LIN {X 0,Y 347.087,Z 840.961,A -85,B 0,C 180,E1 20651.677,E2 20651.677} C_VEL
LIN {X 0,Y 346.368,Z 839.475,A -85,B 0,C 180,E1 20653.232,E2 20653.232} C_VEL
LIN {X 0,Y 343.386,Z 836.917,A -85,B 0,C 180,E1 20663.758,E2 20663.758} C_VEL
LIN {X 0,Y 344.875,Z 838.107,A -85,B 0,C 180,E1 20672.864,E2 20672.864} C_VEL
LIN {X 0,Y 348.52,Z 840.648,A -85,B 0,C 180,E1 20679.253,E2 20679.253} C_VEL
LIN {X 0,Y 352.329,Z 846.298,A -85,B 0,C 180,E1 20684.292,E2 20684.292} C_VEL
LIN {X 0,Y 354.573,Z 848.436,A -85,B 0,C 180,E1 20686.475,E2 20686.475} C_VEL
LIN {X 0,Y 359.696,Z 854.398,A -85,B 0,C 180,E1 20690.882,E2 20690.882} C_VEL
LIN {X 0,Y 364.724,Z 861.307,A -85,B 0,C 180,E1 20694.66,E2 20694.66} C_VEL
LIN {X 0,Y 374.327,Z 875.302,A -85,B 0,C 180,E1 20700.736,E2 20700.736} C_VEL
LIN {X 0,Y 387.121,Z 895.572,A -85,B 0,C 180,E1 20707.425,E2 20707.425} C_VEL
LIN {X 0,Y 401.281,Z 919.676,A -85,B 0,C 180,E1 20713.739,E2 20713.739} C_VEL
LIN {X 0,Y 415.418,Z 946.976,A -85,B 0,C 180,E1 20719.523,E2 20719.523} C_VEL
LIN {X 0,Y 429.203,Z 977.889,A -85,B 0,C 180,E1 20724.99,E2 20724.99} C_VEL
LIN {X 0,Y 433.479,Z 989.391,A -85,B 0,C 180,E1 20726.807,E2 20726.807} C_VEL
LIN {X 0,Y 418.447,Z 1036.021,A -85,B 0,C 180,E1 20729.455,E2 20729.455} C_VEL
LIN {X 0,Y 400.123,Z 1083.411,A -85,B 0,C 180,E1 20733.256,E2 20733.256} C_VEL
LIN {X 0,Y 383.119,Z 1122.716,A -85,B 0,C 180,E1 20737.596,E2 20737.596} C_VEL
LIN {X 0,Y 366.033,Z 1159.658,A -85,B 0,C 180,E1 20743.097,E2 20743.097} C_VEL
LIN {X 0,Y 351.513,Z 1190.56,A -85,B 0,C 180,E1 20749.344,E2 20749.344} C_VEL
LIN {X 0,Y 339.716,Z 1217.292,A -85,B 0,C 180,E1 20756.591,E2 20756.591} C_VEL
LIN {X 0,Y 331.936,Z 1238.037,A -85,B 0,C 180,E1 20764.364,E2 20764.364} C_VEL
LIN {X 0,Y 328.007,Z 1253.422,A -85,B 0,C 180,E1 20772.565,E2 20772.565} C_VEL
LIN {X 0,Y 326.864,Z 1261.496,A -85,B 0,C 180,E1 20779.333,E2 20779.333} C_VEL
LIN {X 0,Y 326.773,Z 1264.976,A -85,B 0,C 180,E1 20784.683,E2 20784.683} C_VEL
LIN {X 0,Y 327.283,Z 1265.936,A -85,B 0,C 180,E1 20789.989,E2 20789.989} C_VEL
LIN {X 0,Y 327.033,Z 1263.961,A -85,B 0,C 180,E1 20795.291,E2 20795.291} C_VEL
LIN {X 0,Y 327.282,Z 1257.785,A -85,B 0,C 180,E1 20801.98,E2 20801.98} C_VEL
LIN {X 0,Y 328.698,Z 1247.276,A -85,B 0,C 180,E1 20808.76,E2 20808.76} C_VEL
LIN {X 0,Y 333.133,Z 1228.55,A -85,B 0,C 180,E1 20816.962,E2 20816.962} C_VEL
LIN {X 0,Y 340.815,Z 1205.172,A -85,B 0,C 180,E1 20824.41,E2 20824.41} C_VEL
LIN {X 0,Y 352.574,Z 1174.665,A -85,B 0,C 180,E1 20831.655,E2 20831.655} C_VEL
LIN {X 0,Y 369.605,Z 1134.827,A -85,B 0,C 180,E1 20838.789,E2 20838.789} C_VEL
LIN {X 0,Y 399.925,Z 1072.683,A -85,B 0,C 180,E1 20846.92,E2 20846.92} C_VEL
LIN {X 0,Y 420.751,Z 1039.494,A -85,B 0,C 180,E1 20850.42,E2 20850.42} C_VEL
LIN {X 0,Y 414.218,Z 1046.912,A -85,B 0,C 180,E1 20851.536,E2 20851.536} C_VEL
LIN {X 0,Y 403.987,Z 1058.605,A -85,B 0,C 180,E1 20852.711,E2 20852.711} C_VEL
LIN {X 0,Y 393.91,Z 1069.679,A -85,B 0,C 180,E1 20853.981,E2 20853.981} C_VEL
LIN {X 0,Y 366.198,Z 1101.609,A -85,B 0,C 180,E1 20861.35,E2 20861.35} C_VEL
LIN {X 0,Y 346.971,Z 1124.322,A -85,B 0,C 180,E1 20868.879,E2 20868.879} C_VEL
LIN {X 0,Y 332.663,Z 1141.932,A -85,B 0,C 180,E1 20877.586,E2 20877.586} C_VEL
LIN {X 0,Y 324.133,Z 1153.386,A -85,B 0,C 180,E1 20886.691,E2 20886.691} C_VEL
LIN {X 0,Y 320.638,Z 1158.38,A -85,B 0,C 180,E1 20893.627,E2 20893.627} C_VEL
LIN {X 0,Y 318.865,Z 1160.285,A -85,B 0,C 180,E1 20899.371,E2 20899.371} C_VEL
LIN {X 0,Y 318.24,Z 1159.445,A -85,B 0,C 180,E1 20908.345,E2 20908.345} C_VEL
LIN {X 0,Y 320.177,Z 1153.951,A -85,B 0,C 180,E1 20916.668,E2 20916.668} C_VEL
LIN {X 0,Y 323.485,Z 1144.81,A -85,B 0,C 180,E1 20924.477,E2 20924.477} C_VEL
LIN {X 0,Y 330.102,Z 1130.596,A -85,B 0,C 180,E1 20932.434,E2 20932.434} C_VEL
LIN {X 0,Y 341.206,Z 1109.637,A -85,B 0,C 180,E1 20940.43,E2 20940.43} C_VEL
LIN {X 0,Y 354.83,Z 1084.984,A -85,B 0,C 180,E1 20947.16,E2 20947.16} C_VEL
LIN {X 0,Y 371.931,Z 1052.972,A -85,B 0,C 180,E1 20953.488,E2 20953.488} C_VEL
LIN {X 0,Y 389.199,Z 1018.22,A -85,B 0,C 180,E1 20958.439,E2 20958.439} C_VEL
LIN {X 0,Y 402.022,Z 989.391,A -85,B 0,C 180,E1 20961.634,E2 20961.634} C_VEL
LIN {X 0,Y 397.777,Z 963.333,A -85,B 0,C 180,E1 20967.015,E2 20967.015} C_VEL
LIN {X 0,Y 391.25,Z 938.761,A -85,B 0,C 180,E1 20972.5,E2 20972.5} C_VEL
LIN {X 0,Y 383.479,Z 917.337,A -85,B 0,C 180,E1 20978.002,E2 20978.002} C_VEL
LIN {X 0,Y 374.105,Z 897.059,A -85,B 0,C 180,E1 20984.227,E2 20984.227} C_VEL
LIN {X 0,Y 364.994,Z 880.396,A -85,B 0,C 180,E1 20990.659,E2 20990.659} C_VEL
LIN {X 0,Y 356.896,Z 867.057,A -85,B 0,C 180,E1 20997.245,E2 20997.245} C_VEL
LIN {X 0,Y 351.496,Z 859.187,A -85,B 0,C 180,E1 21002.484,E2 21002.484} C_VEL
LIN {X 0,Y 348.543,Z 853.905,A -85,B 0,C 180,E1 21006.187,E2 21006.187} C_VEL
LIN {X 0,Y 344.933,Z 848.047,A -85,B 0,C 180,E1 21012.142,E2 21012.142} C_VEL
LIN {X 0,Y 341.412,Z 844.833,A -85,B 0,C 180,E1 21022.14,E2 21022.14} C_VEL
LIN {X 0,Y 342.46,Z 845.304,A -85,B 0,C 180,E1 21030.967,E2 21030.967} C_VEL
LIN {X 0,Y 346.658,Z 848.318,A -85,B 0,C 180,E1 21039.063,E2 21039.063} C_VEL
LIN {X 0,Y 350.624,Z 854.035,A -85,B 0,C 180,E1 21044.381,E2 21044.381} C_VEL
LIN {X 0,Y 352.591,Z 856.228,A -85,B 0,C 180,E1 21046.368,E2 21046.368} C_VEL
LIN {X 0,Y 358.34,Z 863.911,A -85,B 0,C 180,E1 21051.519,E2 21051.519} C_VEL
LIN {X 0,Y 364.09,Z 871.747,A -85,B 0,C 180,E1 21055.711,E2 21055.711} C_VEL
LIN {X 0,Y 371.715,Z 882.573,A -85,B 0,C 180,E1 21060.438,E2 21060.438} C_VEL
LIN {X 0,Y 384.55,Z 903.458,A -85,B 0,C 180,E1 21067.385,E2 21067.385} C_VEL
LIN {X 0,Y 398.907,Z 928.625,A -85,B 0,C 180,E1 21073.974,E2 21073.974} C_VEL
LIN {X 0,Y 413.219,Z 957.636,A -85,B 0,C 180,E1 21080.049,E2 21080.049} C_VEL
LIN {X 0,Y 426.149,Z 988.884,A -85,B 0,C 180,E1 21085.549,E2 21085.549} C_VEL
LIN {X 0,Y 427.428,Z 992.49,A -85,B 0,C 180,E1 21086.118,E2 21086.118} C_VEL
LIN {X 0,Y 411.898,Z 1039.158,A -85,B 0,C 180,E1 21088.873,E2 21088.873} C_VEL
LIN {X 0,Y 393.65,Z 1085.05,A -85,B 0,C 180,E1 21092.623,E2 21092.623} C_VEL
LIN {X 0,Y 375.324,Z 1125.898,A -85,B 0,C 180,E1 21097.294,E2 21097.294} C_VEL
LIN {X 0,Y 358.404,Z 1161.367,A -85,B 0,C 180,E1 21102.774,E2 21102.774} C_VEL
LIN {X 0,Y 342.557,Z 1194.163,A -85,B 0,C 180,E1 21109.732,E2 21109.732} C_VEL
LIN {X 0,Y 330.876,Z 1219.831,A -85,B 0,C 180,E1 21117.202,E2 21117.202} C_VEL
LIN {X 0,Y 323.159,Z 1240.493,A -85,B 0,C 180,E1 21125.553,E2 21125.553} C_VEL
LIN {X 0,Y 319.856,Z 1253.989,A -85,B 0,C 180,E1 21133.522,E2 21133.522} C_VEL
LIN {X 0,Y 318.936,Z 1261.313,A -85,B 0,C 180,E1 21140.444,E2 21140.444} C_VEL
LIN {X 0,Y 319.149,Z 1264.519,A -85,B 0,C 180,E1 21147.275,E2 21147.275} C_VEL
LIN {X 0,Y 319.396,Z 1263.956,A -85,B 0,C 180,E1 21152.701,E2 21152.701} C_VEL
LIN {X 0,Y 319.221,Z 1259.367,A -85,B 0,C 180,E1 21159.525,E2 21159.525} C_VEL
LIN {X 0,Y 320.143,Z 1250.527,A -85,B 0,C 180,E1 21166.439,E2 21166.439} C_VEL
LIN {X 0,Y 323.154,Z 1235.77,A -85,B 0,C 180,E1 21174.064,E2 21174.064} C_VEL
LIN {X 0,Y 329.761,Z 1214.688,A -85,B 0,C 180,E1 21181.895,E2 21181.895} C_VEL
LIN {X 0,Y 340.513,Z 1186.665,A -85,B 0,C 180,E1 21189.562,E2 21189.562} C_VEL
LIN {X 0,Y 356.571,Z 1149.838,A -85,B 0,C 180,E1 21197.099,E2 21197.099} C_VEL
LIN {X 0,Y 379.459,Z 1102.791,A -85,B 0,C 180,E1 21204.273,E2 21204.273} C_VEL
LIN {X 0,Y 407.74,Z 1056.018,A -85,B 0,C 180,E1 21209.875,E2 21209.875} C_VEL
LIN {X 0,Y 411.948,Z 1050.22,A -85,B 0,C 180,E1 21210.575,E2 21210.575} C_VEL
LIN {X 0,Y 393.91,Z 1069.679,A -85,B 0,C 180,E1 21213.981,E2 21213.981} C_VEL
LIN {X 0,Y 383.621,Z 1080.519,A -85,B 0,C 180,E1 21215.383,E2 21215.383} C_VEL
LIN {X 0,Y 373.62,Z 1090.572,A -85,B 0,C 180,E1 21216.898,E2 21216.898} C_VEL
LIN {X 0,Y 348.296,Z 1118.195,A -85,B 0,C 180,E1 21224.912,E2 21224.912} C_VEL
LIN {X 0,Y 330.88,Z 1137.842,A -85,B 0,C 180,E1 21233.444,E2 21233.444} C_VEL
LIN {X 0,Y 319.47,Z 1151.446,A -85,B 0,C 180,E1 21242.71,E2 21242.71} C_VEL
LIN {X 0,Y 313.933,Z 1158.619,A -85,B 0,C 180,E1 21251.099,E2 21251.099} C_VEL
LIN {X 0,Y 311.719,Z 1161.251,A -85,B 0,C 180,E1 21256.907,E2 21256.907} C_VEL
LIN {X 0,Y 310.439,Z 1161.855,A -85,B 0,C 180,E1 21262.915,E2 21262.915} C_VEL
LIN {X 0,Y 310.489,Z 1160.35,A -85,B 0,C 180,E1 21269.119,E2 21269.119} C_VEL
LIN {X 0,Y 312.034,Z 1156.411,A -85,B 0,C 180,E1 21275.526,E2 21275.526} C_VEL
LIN {X 0,Y 314.99,Z 1148.284,A -85,B 0,C 180,E1 21283.171,E2 21283.171} C_VEL
LIN {X 0,Y 321.499,Z 1134.063,A -85,B 0,C 180,E1 21291.803,E2 21291.803} C_VEL
LIN {X 0,Y 331.447,Z 1115.81,A -85,B 0,C 180,E1 21299.382,E2 21299.382} C_VEL
LIN {X 0,Y 345.916,Z 1090.359,A -85,B 0,C 180,E1 21306.861,E2 21306.861} C_VEL
LIN {X 0,Y 361.451,Z 1062.441,A -85,B 0,C 180,E1 21312.786,E2 21312.786} C_VEL
LIN {X 0,Y 379.966,Z 1026.941,A -85,B 0,C 180,E1 21318.283,E2 21318.283} C_VEL
LIN {X 0,Y 395.881,Z 992.175,A -85,B 0,C 180,E1 21322.332,E2 21322.332} C_VEL
LIN {X 0,Y 391.593,Z 965.019,A -85,B 0,C 180,E1 21328.089,E2 21328.089} C_VEL
LIN {X 0,Y 385.246,Z 941.027,A -85,B 0,C 180,E1 21333.664,E2 21333.664} C_VEL
LIN {X 0,Y 377.827,Z 920.469,A -85,B 0,C 180,E1 21339.215,E2 21339.215} C_VEL
LIN {X 0,Y 368.976,Z 901.092,A -85,B 0,C 180,E1 21345.448,E2 21345.448} C_VEL
LIN {X 0,Y 360.705,Z 885.967,A -85,B 0,C 180,E1 21351.602,E2 21351.602} C_VEL
LIN {X 0,Y 353.28,Z 873.457,A -85,B 0,C 180,E1 21358.077,E2 21358.077} C_VEL
LIN {X 0,Y 348.747,Z 866.385,A -85,B 0,C 180,E1 21362.781,E2 21362.781} C_VEL
LIN {X 0,Y 345.909,Z 861.286,A -85,B 0,C 180,E1 21366.567,E2 21366.567} C_VEL
LIN {X 0,Y 342.565,Z 855.118,A -85,B 0,C 180,E1 21372.576,E2 21372.576} C_VEL
LIN {X 0,Y 339.4,Z 852.307,A -85,B 0,C 180,E1 21383.279,E2 21383.279} C_VEL
LIN {X 0,Y 340.932,Z 853.277,A -85,B 0,C 180,E1 21392.449,E2 21392.449} C_VEL
LIN {X 0,Y 344.532,Z 855.901,A -85,B 0,C 180,E1 21398.888,E2 21398.888} C_VEL
LIN {X 0,Y 348.882,Z 861.791,A -85,B 0,C 180,E1 21404.62,E2 21404.62} C_VEL
LIN {X 0,Y 355.837,Z 871.057,A -85,B 0,C 180,E1 21411.147,E2 21411.147} C_VEL
LIN {X 0,Y 361.762,Z 879.343,A -85,B 0,C 180,E1 21415.558,E2 21415.558} C_VEL
LIN {X 0,Y 368.908,Z 889.842,A -85,B 0,C 180,E1 21420.192,E2 21420.192} C_VEL
LIN {X 0,Y 380.831,Z 909.583,A -85,B 0,C 180,E1 21426.837,E2 21426.837} C_VEL
LIN {X 0,Y 394.818,Z 934.761,A -85,B 0,C 180,E1 21433.558,E2 21433.558} C_VEL
LIN {X 0,Y 408.62,Z 963.621,A -85,B 0,C 180,E1 21439.721,E2 21439.721} C_VEL
LIN {X 0,Y 420.981,Z 994.25,A -85,B 0,C 180,E1 21445.194,E2 21445.194} C_VEL
LIN {X 0,Y 421.256,Z 997.281,A -85,B 0,C 180,E1 21445.548,E2 21445.548} C_VEL
LIN {X 0,Y 404.179,Z 1045.484,A -85,B 0,C 180,E1 21448.513,E2 21448.513} C_VEL
LIN {X 0,Y 386.677,Z 1087.571,A -85,B 0,C 180,E1 21452.085,E2 21452.085} C_VEL
LIN {X 0,Y 367.331,Z 1129.407,A -85,B 0,C 180,E1 21457.017,E2 21457.017} C_VEL
LIN {X 0,Y 349.86,Z 1164.557,A -85,B 0,C 180,E1 21462.743,E2 21462.743} C_VEL
LIN {X 0,Y 334.671,Z 1195.273,A -85,B 0,C 180,E1 21469.517,E2 21469.517} C_VEL
LIN {X 0,Y 322.452,Z 1221.324,A -85,B 0,C 180,E1 21477.51,E2 21477.51} C_VEL
LIN {X 0,Y 315.188,Z 1240.426,A -85,B 0,C 180,E1 21485.625,E2 21485.625} C_VEL
LIN {X 0,Y 312.107,Z 1252.616,A -85,B 0,C 180,E1 21493.101,E2 21493.101} C_VEL
LIN {X 0,Y 311.126,Z 1259.993,A -85,B 0,C 180,E1 21500.202,E2 21500.202} C_VEL
LIN {X 0,Y 311.355,Z 1263.22,A -85,B 0,C 180,E1 21507.207,E2 21507.207} C_VEL
LIN {X 0,Y 311.589,Z 1262.619,A -85,B 0,C 180,E1 21512.768,E2 21512.768} C_VEL
LIN {X 0,Y 311.402,Z 1258.01,A -85,B 0,C 180,E1 21519.767,E2 21519.767} C_VEL
LIN {X 0,Y 312.394,Z 1249.057,A -85,B 0,C 180,E1 21526.859,E2 21526.859} C_VEL
LIN {X 0,Y 315.765,Z 1233.745,A -85,B 0,C 180,E1 21534.897,E2 21534.897} C_VEL
LIN {X 0,Y 323.109,Z 1211.687,A -85,B 0,C 180,E1 21543.164,E2 21543.164} C_VEL
LIN {X 0,Y 335.24,Z 1182.08,A -85,B 0,C 180,E1 21551.225,E2 21551.225} C_VEL
LIN {X 0,Y 353.239,Z 1143.875,A -85,B 0,C 180,E1 21558.984,E2 21558.984} C_VEL
LIN {X 0,Y 386.251,Z 1084.14,A -85,B 0,C 180,E1 21567.804,E2 21567.804} C_VEL
LIN {X 0,Y 401.734,Z 1062.211,A -85,B 0,C 180,E1 21570.426,E2 21570.426} C_VEL
LIN {X 0,Y 402.585,Z 1060.814,A -85,B 0,C 180,E1 21570.795,E2 21570.795} C_VEL
LIN {X 0,Y 373.62,Z 1090.572,A -85,B 0,C 180,E1 21576.898,E2 21576.898} C_VEL
LIN {X 0,Y 363.497,Z 1100.296,A -85,B 0,C 180,E1 21578.545,E2 21578.545} C_VEL
LIN {X 0,Y 353.613,Z 1109.353,A -85,B 0,C 180,E1 21580.331,E2 21580.331} C_VEL
LIN {X 0,Y 330.859,Z 1132.881,A -85,B 0,C 180,E1 21589.139,E2 21589.139} C_VEL
LIN {X 0,Y 315.905,Z 1148.961,A -85,B 0,C 180,E1 21598.629,E2 21598.629} C_VEL
LIN {X 0,Y 308.444,Z 1157.652,A -85,B 0,C 180,E1 21607.034,E2 21607.034} C_VEL
LIN {X 0,Y 304.794,Z 1161.898,A -85,B 0,C 180,E1 21614.35,E2 21614.35} C_VEL
LIN {X 0,Y 303.041,Z 1163.313,A -85,B 0,C 180,E1 21620.427,E2 21620.427} C_VEL
LIN {X 0,Y 302.488,Z 1162.504,A -85,B 0,C 180,E1 21626.715,E2 21626.715} C_VEL
LIN {X 0,Y 304.202,Z 1157.914,A -85,B 0,C 180,E1 21635.368,E2 21635.368} C_VEL
LIN {X 0,Y 307.365,Z 1149.485,A -85,B 0,C 180,E1 21643.489,E2 21643.489} C_VEL
LIN {X 0,Y 314.347,Z 1134.909,A -85,B 0,C 180,E1 21652.461,E2 21652.461} C_VEL
LIN {X 0,Y 324.691,Z 1116.522,A -85,B 0,C 180,E1 21660.166,E2 21660.166} C_VEL
LIN {X 0,Y 340.239,Z 1090.054,A -85,B 0,C 180,E1 21667.952,E2 21667.952} C_VEL
LIN {X 0,Y 357.448,Z 1059.64,A -85,B 0,C 180,E1 21674.285,E2 21674.285} C_VEL
LIN {X 0,Y 375.839,Z 1025.164,A -85,B 0,C 180,E1 21679.498,E2 21679.498} C_VEL
LIN {X 0,Y 389.627,Z 996.191,A -85,B 0,C 180,E1 21682.818,E2 21682.818} C_VEL
LIN {X 0,Y 386.32,Z 971.848,A -85,B 0,C 180,E1 21688.048,E2 21688.048} C_VEL
LIN {X 0,Y 380.76,Z 948.316,A -85,B 0,C 180,E1 21693.611,E2 21693.611} C_VEL
LIN {X 0,Y 374,Z 928.346,A -85,B 0,C 180,E1 21699.017,E2 21699.017} C_VEL
LIN {X 0,Y 365.792,Z 909.081,A -85,B 0,C 180,E1 21705.256,E2 21705.256} C_VEL
LIN {X 0,Y 357.652,Z 893.36,A -85,B 0,C 180,E1 21711.654,E2 21711.654} C_VEL
LIN {X 0,Y 350.277,Z 880.59,A -85,B 0,C 180,E1 21718.34,E2 21718.34} C_VEL
LIN {X 0,Y 346.244,Z 873.969,A -85,B 0,C 180,E1 21722.707,E2 21722.707} C_VEL
LIN {X 0,Y 344.049,Z 869.094,A -85,B 0,C 180,E1 21725.952,E2 21725.952} C_VEL
LIN {X 0,Y 340.256,Z 863.172,A -85,B 0,C 180,E1 21732.426,E2 21732.426} C_VEL
LIN {X 0,Y 337.277,Z 860.03,A -85,B 0,C 180,E1 21742.323,E2 21742.323} C_VEL
LIN {X 0,Y 338.315,Z 860.479,A -85,B 0,C 180,E1 21750.576,E2 21750.576} C_VEL
LIN {X 0,Y 342.401,Z 863.472,A -85,B 0,C 180,E1 21758.697,E2 21758.697} C_VEL
LIN {X 0,Y 346.957,Z 869.474,A -85,B 0,C 180,E1 21764.693,E2 21764.693} C_VEL
LIN {X 0,Y 353.516,Z 878.724,A -85,B 0,C 180,E1 21771.037,E2 21771.037} C_VEL
LIN {X 0,Y 359.005,Z 886.571,A -85,B 0,C 180,E1 21775.303,E2 21775.303} C_VEL
LIN {X 0,Y 366.202,Z 897.441,A -85,B 0,C 180,E1 21780.045,E2 21780.045} C_VEL
LIN {X 0,Y 377.529,Z 916.653,A -85,B 0,C 180,E1 21786.605,E2 21786.605} C_VEL
LIN {X 0,Y 390.304,Z 940.278,A -85,B 0,C 180,E1 21793.006,E2 21793.006} C_VEL
LIN {X 0,Y 403.47,Z 968.31,A -85,B 0,C 180,E1 21799.129,E2 21799.129} C_VEL
LIN {X 0,Y 415.487,Z 998.842,A -85,B 0,C 180,E1 21804.722,E2 21804.722} C_VEL
LIN {X 0,Y 397.445,Z 1049.215,A -85,B 0,C 180,E1 21807.946,E2 21807.946} C_VEL
LIN {X 0,Y 378.508,Z 1092.765,A -85,B 0,C 180,E1 21811.823,E2 21811.823} C_VEL
LIN {X 0,Y 360.009,Z 1131.337,A -85,B 0,C 180,E1 21816.538,E2 21816.538} C_VEL
LIN {X 0,Y 341.309,Z 1167.786,A -85,B 0,C 180,E1 21822.719,E2 21822.719} C_VEL
LIN {X 0,Y 326.235,Z 1197.103,A -85,B 0,C 180,E1 21829.561,E2 21829.561} C_VEL
LIN {X 0,Y 314.599,Z 1221.479,A -85,B 0,C 180,E1 21837.347,E2 21837.347} C_VEL
LIN {X 0,Y 307.118,Z 1240.519,A -85,B 0,C 180,E1 21845.878,E2 21845.878} C_VEL
LIN {X 0,Y 304.013,Z 1252.978,A -85,B 0,C 180,E1 21854.123,E2 21854.123} C_VEL
LIN {X 0,Y 303.306,Z 1259.571,A -85,B 0,C 180,E1 21861.393,E2 21861.393} C_VEL
LIN {X 0,Y 303.552,Z 1261.917,A -85,B 0,C 180,E1 21867.135,E2 21867.135} C_VEL
LIN {X 0,Y 303.789,Z 1261.304,A -85,B 0,C 180,E1 21872.839,E2 21872.839} C_VEL
LIN {X 0,Y 303.59,Z 1256.617,A -85,B 0,C 180,E1 21880.021,E2 21880.021} C_VEL
LIN {X 0,Y 304.642,Z 1247.636,A -85,B 0,C 180,E1 21887.302,E2 21887.302} C_VEL
LIN {X 0,Y 308.316,Z 1232.045,A -85,B 0,C 180,E1 21895.633,E2 21895.633} C_VEL
LIN {X 0,Y 316.164,Z 1209.949,A -85,B 0,C 180,E1 21904.065,E2 21904.065} C_VEL
LIN {X 0,Y 328.522,Z 1181.375,A -85,B 0,C 180,E1 21912.04,E2 21912.04} C_VEL
LIN {X 0,Y 348.658,Z 1141.259,A -85,B 0,C 180,E1 21920.351,E2 21920.351} C_VEL
LIN {X 0,Y 384.664,Z 1082.472,A -85,B 0,C 180,E1 21929.231,E2 21929.231} C_VEL
LIN {X 0,Y 394.161,Z 1069.933,A -85,B 0,C 180,E1 21930.852,E2 21930.852} C_VEL
LIN {X 0,Y 359.944,Z 1102.999,A -85,B 0,C 180,E1 21938.449,E2 21938.449} C_VEL
LIN {X 0,Y 353.613,Z 1109.353,A -85,B 0,C 180,E1 21940.331,E2 21940.331} C_VEL
LIN {X 0,Y 343.732,Z 1117.929,A -85,B 0,C 180,E1 21942.253,E2 21942.253} C_VEL
LIN {X 0,Y 334.932,Z 1125.088,A -85,B 0,C 180,E1 21944.007,E2 21944.007} C_VEL
LIN {X 0,Y 334.039,Z 1125.919,A -85,B 0,C 180,E1 21944.318,E2 21944.318} C_VEL
LIN {X 0,Y 315.799,Z 1143.775,A -85,B 0,C 180,E1 21953.129,E2 21953.129} C_VEL
LIN {X 0,Y 305.227,Z 1154.752,A -85,B 0,C 180,E1 21961.417,E2 21961.417} C_VEL
LIN {X 0,Y 299.684,Z 1160.788,A -85,B 0,C 180,E1 21968.699,E2 21968.699} C_VEL
LIN {X 0,Y 295.873,Z 1164.379,A -85,B 0,C 180,E1 21977.842,E2 21977.842} C_VEL
LIN {X 0,Y 294.752,Z 1164.489,A -85,B 0,C 180,E1 21984.21,E2 21984.21} C_VEL
LIN {X 0,Y 295.712,Z 1160.822,A -85,B 0,C 180,E1 21993.059,E2 21993.059} C_VEL
LIN {X 0,Y 298.479,Z 1153.795,A -85,B 0,C 180,E1 22001.153,E2 22001.153} C_VEL
LIN {X 0,Y 304.268,Z 1141.245,A -85,B 0,C 180,E1 22010.22,E2 22010.22} C_VEL
LIN {X 0,Y 314.361,Z 1123.295,A -85,B 0,C 180,E1 22018.663,E2 22018.663} C_VEL
LIN {X 0,Y 327.801,Z 1101.026,A -85,B 0,C 180,E1 22026.118,E2 22026.118} C_VEL
LIN {X 0,Y 345.295,Z 1071.607,A -85,B 0,C 180,E1 22033.056,E2 22033.056} C_VEL
LIN {X 0,Y 363.054,Z 1039.973,A -85,B 0,C 180,E1 22038.461,E2 22038.461} C_VEL
LIN {X 0,Y 382.885,Z 1000.352,A -85,B 0,C 180,E1 22043.352,E2 22043.352} C_VEL
LIN {X 0,Y 383.212,Z 995.088,A -85,B 0,C 180,E1 22044.352,E2 22044.352} C_VEL
LIN {X 0,Y 379.5,Z 970.078,A -85,B 0,C 180,E1 22050.009,E2 22050.009} C_VEL
LIN {X 0,Y 373.682,Z 946.778,A -85,B 0,C 180,E1 22055.812,E2 22055.812} C_VEL
LIN {X 0,Y 366.353,Z 926.234,A -85,B 0,C 180,E1 22061.911,E2 22061.911} C_VEL
LIN {X 0,Y 358.187,Z 907.951,A -85,B 0,C 180,E1 22068.52,E2 22068.52} C_VEL
LIN {X 0,Y 350.102,Z 893.031,A -85,B 0,C 180,E1 22075.58,E2 22075.58} C_VEL
LIN {X 0,Y 344.531,Z 882.474,A -85,B 0,C 180,E1 22081.768,E2 22081.768} C_VEL
LIN {X 0,Y 340.586,Z 875.97,A -85,B 0,C 180,E1 22087.009,E2 22087.009} C_VEL
LIN {X 0,Y 336.681,Z 869.369,A -85,B 0,C 180,E1 22095.184,E2 22095.184} C_VEL
LIN {X 0,Y 335.003,Z 867.381,A -85,B 0,C 180,E1 22104.3,E2 22104.3} C_VEL
LIN {X 0,Y 337.251,Z 868.922,A -85,B 0,C 180,E1 22113.673,E2 22113.673} C_VEL
LIN {X 0,Y 340.17,Z 871.16,A -85,B 0,C 180,E1 22118.626,E2 22118.626} C_VEL
LIN {X 0,Y 345.739,Z 878.913,A -85,B 0,C 180,E1 22125.869,E2 22125.869} C_VEL
LIN {X 0,Y 351.052,Z 886.359,A -85,B 0,C 180,E1 22130.964,E2 22130.964} C_VEL
LIN {X 0,Y 357.173,Z 895.047,A -85,B 0,C 180,E1 22135.679,E2 22135.679} C_VEL
LIN {X 0,Y 366.164,Z 909.503,A -85,B 0,C 180,E1 22141.684,E2 22141.684} C_VEL
LIN {X 0,Y 378.382,Z 931.271,A -85,B 0,C 180,E1 22148.613,E2 22148.613} C_VEL
LIN {X 0,Y 391.23,Z 957.078,A -85,B 0,C 180,E1 22155.112,E2 22155.112} C_VEL
LIN {X 0,Y 403.088,Z 984.709,A -85,B 0,C 180,E1 22160.862,E2 22160.862} C_VEL
LIN {X 0,Y 409.541,Z 1002.363,A -85,B 0,C 180,E1 22164.089,E2 22164.089} C_VEL
LIN {X 0,Y 392.223,Z 1049.016,A -85,B 0,C 180,E1 22167.076,E2 22167.076} C_VEL
LIN {X 0,Y 372.221,Z 1093.846,A -85,B 0,C 180,E1 22171.11,E2 22171.11} C_VEL
LIN {X 0,Y 352.983,Z 1132.522,A -85,B 0,C 180,E1 22175.955,E2 22175.955} C_VEL
LIN {X 0,Y 334.048,Z 1168.48,A -85,B 0,C 180,E1 22182.194,E2 22182.194} C_VEL
LIN {X 0,Y 318.816,Z 1197.067,A -85,B 0,C 180,E1 22189.084,E2 22189.084} C_VEL
LIN {X 0,Y 306.721,Z 1221.592,A -85,B 0,C 180,E1 22197.173,E2 22197.173} C_VEL
LIN {X 0,Y 299.615,Z 1238.973,A -85,B 0,C 180,E1 22205.2,E2 22205.2} C_VEL
LIN {X 0,Y 296.276,Z 1251.58,A -85,B 0,C 180,E1 22213.697,E2 22213.697} C_VEL
LIN {X 0,Y 295.487,Z 1258.232,A -85,B 0,C 180,E1 22221.163,E2 22221.163} C_VEL
LIN {X 0,Y 295.739,Z 1260.598,A -85,B 0,C 180,E1 22227.059,E2 22227.059} C_VEL
LIN {X 0,Y 295.986,Z 1259.967,A -85,B 0,C 180,E1 22232.914,E2 22232.914} C_VEL
LIN {X 0,Y 295.777,Z 1255.228,A -85,B 0,C 180,E1 22240.288,E2 22240.288} C_VEL
LIN {X 0,Y 296.892,Z 1246.194,A -85,B 0,C 180,E1 22247.768,E2 22247.768} C_VEL
LIN {X 0,Y 300.84,Z 1230.591,A -85,B 0,C 180,E1 22256.305,E2 22256.305} C_VEL
LIN {X 0,Y 309.357,Z 1208.015,A -85,B 0,C 180,E1 22265.089,E2 22265.089} C_VEL
LIN {X 0,Y 323.24,Z 1177.994,A -85,B 0,C 180,E1 22273.561,E2 22273.561} C_VEL
LIN {X 0,Y 346.129,Z 1135.75,A -85,B 0,C 180,E1 22282.326,E2 22282.326} C_VEL
LIN {X 0,Y 382.141,Z 1082.912,A -85,B 0,C 180,E1 22290.43,E2 22290.43} C_VEL
LIN {X 0,Y 385.213,Z 1079.225,A -85,B 0,C 180,E1 22290.993,E2 22290.993} C_VEL
LIN {X 0,Y 348.912,Z 1111.82,A -85,B 0,C 180,E1 22299.33,E2 22299.33} C_VEL
LIN {X 0,Y 334.039,Z 1125.919,A -85,B 0,C 180,E1 22304.318,E2 22304.318} C_VEL
LIN {X 0,Y 324.659,Z 1133.289,A -85,B 0,C 180,E1 22306.556,E2 22306.556} C_VEL
LIN {X 0,Y 316.363,Z 1139.374,A -85,B 0,C 180,E1 22308.602,E2 22308.602} C_VEL
LIN {X 0,Y 315.561,Z 1140.044,A -85,B 0,C 180,E1 22308.95,E2 22308.95} C_VEL
LIN {X 0,Y 300.487,Z 1154.13,A -85,B 0,C 180,E1 22318.558,E2 22318.558} C_VEL
LIN {X 0,Y 293.757,Z 1160.823,A -85,B 0,C 180,E1 22325.904,E2 22325.904} C_VEL
LIN {X 0,Y 288.915,Z 1165.306,A -85,B 0,C 180,E1 22335.158,E2 22335.158} C_VEL
LIN {X 0,Y 287.237,Z 1166.01,A -85,B 0,C 180,E1 22341.605,E2 22341.605} C_VEL
LIN {X 0,Y 286.984,Z 1164.651,A -85,B 0,C 180,E1 22348.284,E2 22348.284} C_VEL
LIN {X 0,Y 288.844,Z 1159.754,A -85,B 0,C 180,E1 22356.428,E2 22356.428} C_VEL
LIN {X 0,Y 292.425,Z 1151.074,A -85,B 0,C 180,E1 22364.778,E2 22364.778} C_VEL
LIN {X 0,Y 299.918,Z 1136.859,A -85,B 0,C 180,E1 22373.713,E2 22373.713} C_VEL
LIN {X 0,Y 311.248,Z 1118.044,A -85,B 0,C 180,E1 22381.752,E2 22381.752} C_VEL
LIN {X 0,Y 327.464,Z 1092.142,A -85,B 0,C 180,E1 22389.53,E2 22389.53} C_VEL
LIN {X 0,Y 345.244,Z 1062.316,A -85,B 0,C 180,E1 22395.856,E2 22395.856} C_VEL
LIN {X 0,Y 364.991,Z 1026.902,A -85,B 0,C 180,E1 22401.276,E2 22401.276} C_VEL
LIN {X 0,Y 377.391,Z 1001.618,A -85,B 0,C 180,E1 22404.265,E2 22404.265} C_VEL
LIN {X 0,Y 374.238,Z 976.665,A -85,B 0,C 180,E1 22410.009,E2 22410.009} C_VEL
LIN {X 0,Y 369.108,Z 953.674,A -85,B 0,C 180,E1 22415.862,E2 22415.862} C_VEL
LIN {X 0,Y 362.66,Z 934.366,A -85,B 0,C 180,E1 22421.609,E2 22421.609} C_VEL
LIN {X 0,Y 355.156,Z 916.467,A -85,B 0,C 180,E1 22428.041,E2 22428.041} C_VEL
LIN {X 0,Y 347.533,Z 901.223,A -85,B 0,C 180,E1 22435.079,E2 22435.079} C_VEL
LIN {X 0,Y 341.354,Z 889.501,A -85,B 0,C 180,E1 22442.098,E2 22442.098} C_VEL
LIN {X 0,Y 338.376,Z 883.895,A -85,B 0,C 180,E1 22446.51,E2 22446.51} C_VEL
LIN {X 0,Y 334.713,Z 877.476,A -85,B 0,C 180,E1 22453.758,E2 22453.758} C_VEL
LIN {X 0,Y 332.741,Z 874.964,A -85,B 0,C 180,E1 22463.82,E2 22463.82} C_VEL
LIN {X 0,Y 334.732,Z 876.279,A -85,B 0,C 180,E1 22473.167,E2 22473.167} C_VEL
LIN {X 0,Y 337.727,Z 878.651,A -85,B 0,C 180,E1 22478.434,E2 22478.434} C_VEL
LIN {X 0,Y 343.18,Z 886.317,A -85,B 0,C 180,E1 22485.662,E2 22485.662} C_VEL
LIN {X 0,Y 348.551,Z 893.884,A -85,B 0,C 180,E1 22490.842,E2 22490.842} C_VEL
LIN {X 0,Y 356.46,Z 905.399,A -85,B 0,C 180,E1 22496.964,E2 22496.964} C_VEL
LIN {X 0,Y 367.298,Z 924.206,A -85,B 0,C 180,E1 22504.046,E2 22504.046} C_VEL
LIN {X 0,Y 379.521,Z 947.472,A -85,B 0,C 180,E1 22510.902,E2 22510.902} C_VEL
LIN {X 0,Y 391.999,Z 974.969,A -85,B 0,C 180,E1 22517.382,E2 22517.382} C_VEL
LIN {X 0,Y 402.866,Z 1003.488,A -85,B 0,C 180,E1 22523.007,E2 22523.007} C_VEL
LIN {X 0,Y 403.595,Z 1005.65,A -85,B 0,C 180,E1 22523.401,E2 22523.401} C_VEL
LIN {X 0,Y 386.456,Z 1050.089,A -85,B 0,C 180,E1 22526.298,E2 22526.298} C_VEL
LIN {X 0,Y 365.255,Z 1096.414,A -85,B 0,C 180,E1 22530.54,E2 22530.54} C_VEL
LIN {X 0,Y 345.78,Z 1134.145,A -85,B 0,C 180,E1 22535.417,E2 22535.417} C_VEL
LIN {X 0,Y 326.569,Z 1169.422,A -85,B 0,C 180,E1 22541.729,E2 22541.729} C_VEL
LIN {X 0,Y 309.773,Z 1200.109,A -85,B 0,C 180,E1 22549.482,E2 22549.482} C_VEL
LIN {X 0,Y 297.919,Z 1223.527,A -85,B 0,C 180,E1 22557.807,E2 22557.807} C_VEL
LIN {X 0,Y 290.712,Z 1241.694,A -85,B 0,C 180,E1 22567.043,E2 22567.043} C_VEL
LIN {X 0,Y 288.238,Z 1251.898,A -85,B 0,C 180,E1 22574.792,E2 22574.792} C_VEL
LIN {X 0,Y 287.692,Z 1256.882,A -85,B 0,C 180,E1 22580.922,E2 22580.922} C_VEL
LIN {X 0,Y 287.935,Z 1259.269,A -85,B 0,C 180,E1 22586.98,E2 22586.98} C_VEL
LIN {X 0,Y 288.182,Z 1258.621,A -85,B 0,C 180,E1 22592.993,E2 22592.993} C_VEL
LIN {X 0,Y 287.965,Z 1253.88,A -85,B 0,C 180,E1 22600.57,E2 22600.57} C_VEL
LIN {X 0,Y 289.173,Z 1244.797,A -85,B 0,C 180,E1 22608.259,E2 22608.259} C_VEL
LIN {X 0,Y 293.418,Z 1229.006,A -85,B 0,C 180,E1 22617.074,E2 22617.074} C_VEL
LIN {X 0,Y 302.349,Z 1206.74,A -85,B 0,C 180,E1 22625.946,E2 22625.946} C_VEL
LIN {X 0,Y 317.304,Z 1176.521,A -85,B 0,C 180,E1 22634.695,E2 22634.695} C_VEL
LIN {X 0,Y 343.355,Z 1131.951,A -85,B 0,C 180,E1 22644.091,E2 22644.091} C_VEL
LIN {X 0,Y 375.945,Z 1088.152,A -85,B 0,C 180,E1 22651.163,E2 22651.163} C_VEL
LIN {X 0,Y 341.176,Z 1117.219,A -85,B 0,C 180,E1 22659.248,E2 22659.248} C_VEL
LIN {X 0,Y 317.601,Z 1138.246,A -85,B 0,C 180,E1 22667.973,E2 22667.973} C_VEL
LIN {X 0,Y 315.561,Z 1140.044,A -85,B 0,C 180,E1 22668.95,E2 22668.95} C_VEL
LIN {X 0,Y 306.786,Z 1146.202,A -85,B 0,C 180,E1 22671.512,E2 22671.512} C_VEL
LIN {X 0,Y 298.45,Z 1151.71,A -85,B 0,C 180,E1 22674.241,E2 22674.241} C_VEL
LIN {X 0,Y 287.652,Z 1161.404,A -85,B 0,C 180,E1 22683.749,E2 22683.749} C_VEL
LIN {X 0,Y 282.29,Z 1166.123,A -85,B 0,C 180,E1 22692.362,E2 22692.362} C_VEL
LIN {X 0,Y 279.335,Z 1167.311,A -85,B 0,C 180,E1 22702.249,E2 22702.249} C_VEL
LIN {X 0,Y 279.961,Z 1163.74,A -85,B 0,C 180,E1 22712.663,E2 22712.663} C_VEL
LIN {X 0,Y 282.366,Z 1158.106,A -85,B 0,C 180,E1 22719.95,E2 22719.95} C_VEL
LIN {X 0,Y 287.254,Z 1147.475,A -85,B 0,C 180,E1 22728.659,E2 22728.659} C_VEL
LIN {X 0,Y 297.072,Z 1130.798,A -85,B 0,C 180,E1 22737.765,E2 22737.765} C_VEL
LIN {X 0,Y 310.702,Z 1109.219,A -85,B 0,C 180,E1 22745.82,E2 22745.82} C_VEL
LIN {X 0,Y 328.11,Z 1081.969,A -85,B 0,C 180,E1 22753.019,E2 22753.019} C_VEL
LIN {X 0,Y 347.086,Z 1050.328,A -85,B 0,C 180,E1 22758.944,E2 22758.944} C_VEL
LIN {X 0,Y 367.216,Z 1013.347,A -85,B 0,C 180,E1 22763.952,E2 22763.952} C_VEL
LIN {X 0,Y 371.243,Z 1004.88,A -85,B 0,C 180,E1 22764.9,E2 22764.9} C_VEL
LIN {X 0,Y 368.551,Z 980.848,A -85,B 0,C 180,E1 22770.597,E2 22770.597} C_VEL
LIN {X 0,Y 364.04,Z 959.179,A -85,B 0,C 180,E1 22776.253,E2 22776.253} C_VEL
LIN {X 0,Y 357.894,Z 939.746,A -85,B 0,C 180,E1 22782.197,E2 22782.197} C_VEL
LIN {X 0,Y 350.872,Z 922.257,A -85,B 0,C 180,E1 22788.669,E2 22788.669} C_VEL
LIN {X 0,Y 344.013,Z 908.084,A -85,B 0,C 180,E1 22795.37,E2 22795.37} C_VEL
LIN {X 0,Y 338.173,Z 896.554,A -85,B 0,C 180,E1 22802.437,E2 22802.437} C_VEL
LIN {X 0,Y 333.763,Z 889.166,A -85,B 0,C 180,E1 22809.346,E2 22809.346} C_VEL
LIN {X 0,Y 332.277,Z 885.37,A -85,B 0,C 180,E1 22813.318,E2 22813.318} C_VEL
LIN {X 0,Y 330.223,Z 882.879,A -85,B 0,C 180,E1 22821.085,E2 22821.085} C_VEL
LIN {X 0,Y 331.272,Z 882.979,A -85,B 0,C 180,E1 22830.093,E2 22830.093} C_VEL
LIN {X 0,Y 334.828,Z 885.109,A -85,B 0,C 180,E1 22837.362,E2 22837.362} C_VEL
LIN {X 0,Y 340.619,Z 893.829,A -85,B 0,C 180,E1 22845.552,E2 22845.552} C_VEL
LIN {X 0,Y 345.646,Z 901.002,A -85,B 0,C 180,E1 22850.566,E2 22850.566} C_VEL
LIN {X 0,Y 353.747,Z 913.232,A -85,B 0,C 180,E1 22856.999,E2 22856.999} C_VEL
LIN {X 0,Y 364.2,Z 931.951,A -85,B 0,C 180,E1 22864.081,E2 22864.081} C_VEL
LIN {X 0,Y 375.595,Z 954.365,A -85,B 0,C 180,E1 22870.724,E2 22870.724} C_VEL
LIN {X 0,Y 387.186,Z 980.73,A -85,B 0,C 180,E1 22877.02,E2 22877.02} C_VEL
LIN {X 0,Y 397.564,Z 1008.686,A -85,B 0,C 180,E1 22882.633,E2 22882.633} C_VEL
LIN {X 0,Y 379.141,Z 1054.761,A -85,B 0,C 180,E1 22885.784,E2 22885.784} C_VEL
LIN {X 0,Y 358.62,Z 1098.16,A -85,B 0,C 180,E1 22889.886,E2 22889.886} C_VEL
LIN {X 0,Y 336.448,Z 1139.771,A -85,B 0,C 180,E1 22895.491,E2 22895.491} C_VEL
LIN {X 0,Y 317.375,Z 1173.379,A -85,B 0,C 180,E1 22901.95,E2 22901.95} C_VEL
LIN {X 0,Y 301.65,Z 1201.256,A -85,B 0,C 180,E1 22909.352,E2 22909.352} C_VEL
LIN {X 0,Y 289.856,Z 1223.886,A -85,B 0,C 180,E1 22917.821,E2 22917.821} C_VEL
LIN {X 0,Y 282.754,Z 1241.453,A -85,B 0,C 180,E1 22927.191,E2 22927.191} C_VEL
LIN {X 0,Y 280.473,Z 1250.455,A -85,B 0,C 180,E1 22934.36,E2 22934.36} C_VEL
LIN {X 0,Y 279.899,Z 1255.509,A -85,B 0,C 180,E1 22940.667,E2 22940.667} C_VEL
LIN {X 0,Y 280.151,Z 1257.919,A -85,B 0,C 180,E1 22946.896,E2 22946.896} C_VEL
LIN {X 0,Y 280.569,Z 1257.985,A -85,B 0,C 180,E1 22949.987,E2 22949.987} C_VEL
LIN {X 0,Y 280.139,Z 1255.931,A -85,B 0,C 180,E1 22956.18,E2 22956.18} C_VEL
LIN {X 0,Y 280.619,Z 1249.182,A -85,B 0,C 180,E1 22964.251,E2 22964.251} C_VEL
LIN {X 0,Y 282.939,Z 1237.154,A -85,B 0,C 180,E1 22972.766,E2 22972.766} C_VEL
LIN {X 0,Y 289.791,Z 1217.905,A -85,B 0,C 180,E1 22982.142,E2 22982.142} C_VEL
LIN {X 0,Y 302.81,Z 1191.014,A -85,B 0,C 180,E1 22991.539,E2 22991.539} C_VEL
LIN {X 0,Y 325.454,Z 1151.92,A -85,B 0,C 180,E1 23001.276,E2 23001.276} C_VEL
LIN {X 0,Y 361.209,Z 1103.076,A -85,B 0,C 180,E1 23010.141,E2 23010.141} C_VEL
LIN {X 0,Y 365.811,Z 1097.841,A -85,B 0,C 180,E1 23010.962,E2 23010.962} C_VEL
LIN {X 0,Y 366.265,Z 1096.956,A -85,B 0,C 180,E1 23011.392,E2 23011.392} C_VEL
LIN {X 0,Y 330.49,Z 1124.932,A -85,B 0,C 180,E1 23020.045,E2 23020.045} C_VEL
LIN {X 0,Y 305.9,Z 1145.426,A -85,B 0,C 180,E1 23029.9,E2 23029.9} C_VEL
LIN {X 0,Y 298.45,Z 1151.71,A -85,B 0,C 180,E1 23034.241,E2 23034.241} C_VEL
LIN {X 0,Y 290.592,Z 1156.592,A -85,B 0,C 180,E1 23037.138,E2 23037.138} C_VEL
LIN {X 0,Y 283.176,Z 1160.829,A -85,B 0,C 180,E1 23040.2,E2 23040.2} C_VEL
LIN {X 0,Y 275.826,Z 1166.733,A -85,B 0,C 180,E1 23049.646,E2 23049.646} C_VEL
LIN {X 0,Y 272.057,Z 1168.916,A -85,B 0,C 180,E1 23059.464,E2 23059.464} C_VEL
LIN {X 0,Y 271.251,Z 1167.657,A -85,B 0,C 180,E1 23066.991,E2 23066.991} C_VEL
LIN {X 0,Y 272.946,Z 1163.187,A -85,B 0,C 180,E1 23075.536,E2 23075.536} C_VEL
LIN {X 0,Y 276.365,Z 1155.483,A -85,B 0,C 180,E1 23083.908,E2 23083.908} C_VEL
LIN {X 0,Y 284.032,Z 1141.203,A -85,B 0,C 180,E1 23093.709,E2 23093.709} C_VEL
LIN {X 0,Y 295.747,Z 1123.058,A -85,B 0,C 180,E1 23102.157,E2 23102.157} C_VEL
LIN {X 0,Y 312.353,Z 1097.89,A -85,B 0,C 180,E1 23110.218,E2 23110.218} C_VEL
LIN {X 0,Y 330.96,Z 1068.847,A -85,B 0,C 180,E1 23116.815,E2 23116.815} C_VEL
LIN {X 0,Y 352.252,Z 1032.502,A -85,B 0,C 180,E1 23122.616,E2 23122.616} C_VEL
LIN {X 0,Y 364.971,Z 1008.426,A -85,B 0,C 180,E1 23125.527,E2 23125.527} C_VEL
LIN {X 0,Y 363.089,Z 986.238,A -85,B 0,C 180,E1 23130.905,E2 23130.905} C_VEL
LIN {X 0,Y 358.705,Z 963.709,A -85,B 0,C 180,E1 23136.913,E2 23136.913} C_VEL
LIN {X 0,Y 352.622,Z 943.627,A -85,B 0,C 180,E1 23143.295,E2 23143.295} C_VEL
LIN {X 0,Y 346.14,Z 927.099,A -85,B 0,C 180,E1 23149.691,E2 23149.691} C_VEL
LIN {X 0,Y 338.948,Z 911.629,A -85,B 0,C 180,E1 23157.451,E2 23157.451} C_VEL
LIN {X 0,Y 334.111,Z 902.258,A -85,B 0,C 180,E1 23163.974,E2 23163.974} C_VEL
LIN {X 0,Y 330.68,Z 896.202,A -85,B 0,C 180,E1 23169.786,E2 23169.786} C_VEL
LIN {X 0,Y 329.5,Z 892.732,A -85,B 0,C 180,E1 23173.477,E2 23173.477} C_VEL
LIN {X 0,Y 327.612,Z 890.265,A -85,B 0,C 180,E1 23181.654,E2 23181.654} C_VEL
LIN {X 0,Y 328.956,Z 890.633,A -85,B 0,C 180,E1 23190.803,E2 23190.803} C_VEL
LIN {X 0,Y 332.126,Z 892.521,A -85,B 0,C 180,E1 23197.168,E2 23197.168} C_VEL
LIN {X 0,Y 337.59,Z 900.67,A -85,B 0,C 180,E1 23205.088,E2 23205.088} C_VEL
LIN {X 0,Y 345.158,Z 911.726,A -85,B 0,C 180,E1 23212.455,E2 23212.455} C_VEL
LIN {X 0,Y 353.099,Z 924.881,A -85,B 0,C 180,E1 23218.697,E2 23218.697} C_VEL
LIN {X 0,Y 364.25,Z 945.662,A -85,B 0,C 180,E1 23226.073,E2 23226.073} C_VEL
LIN {X 0,Y 375.581,Z 970.011,A -85,B 0,C 180,E1 23232.784,E2 23232.784} C_VEL
LIN {X 0,Y 386.188,Z 996.683,A -85,B 0,C 180,E1 23238.832,E2 23238.832} C_VEL
LIN {X 0,Y 391.28,Z 1013.25,A -85,B 0,C 180,E1 23242.03,E2 23242.03} C_VEL
LIN {X 0,Y 370.964,Z 1061.376,A -85,B 0,C 180,E1 23245.408,E2 23245.408} C_VEL
LIN {X 0,Y 350.72,Z 1102.34,A -85,B 0,C 180,E1 23249.511,E2 23249.511} C_VEL
LIN {X 0,Y 329.814,Z 1140.248,A -85,B 0,C 180,E1 23254.761,E2 23254.761} C_VEL
LIN {X 0,Y 309.697,Z 1174.649,A -85,B 0,C 180,E1 23261.561,E2 23261.561} C_VEL
LIN {X 0,Y 293.901,Z 1201.628,A -85,B 0,C 180,E1 23269.025,E2 23269.025} C_VEL
LIN {X 0,Y 281.407,Z 1224.93,A -85,B 0,C 180,E1 23278.173,E2 23278.173} C_VEL
LIN {X 0,Y 274.77,Z 1241.104,A -85,B 0,C 180,E1 23287.345,E2 23287.345} C_VEL
LIN {X 0,Y 272.414,Z 1250.727,A -85,B 0,C 180,E1 23295.69,E2 23295.69} C_VEL
LIN {X 0,Y 272.091,Z 1255.731,A -85,B 0,C 180,E1 23303.61,E2 23303.61} C_VEL
LIN {X 0,Y 272.801,Z 1256.665,A -85,B 0,C 180,E1 23309.987,E2 23309.987} C_VEL
LIN {X 0,Y 272.34,Z 1254.595,A -85,B 0,C 180,E1 23316.358,E2 23316.358} C_VEL
LIN {X 0,Y 272.821,Z 1247.809,A -85,B 0,C 180,E1 23324.667,E2 23324.667} C_VEL
LIN {X 0,Y 275.344,Z 1235.767,A -85,B 0,C 180,E1 23333.431,E2 23333.431} C_VEL
LIN {X 0,Y 282.625,Z 1216.61,A -85,B 0,C 180,E1 23343.015,E2 23343.015} C_VEL
LIN {X 0,Y 296.462,Z 1189.807,A -85,B 0,C 180,E1 23352.636,E2 23352.636} C_VEL
LIN {X 0,Y 320.902,Z 1150.652,A -85,B 0,C 180,E1 23362.644,E2 23362.644} C_VEL
LIN {X 0,Y 357.185,Z 1105.429,A -85,B 0,C 180,E1 23371.157,E2 23371.157} C_VEL
LIN {X 0,Y 358.171,Z 1104.365,A -85,B 0,C 180,E1 23371.327,E2 23371.327} C_VEL
LIN {X 0,Y 318.578,Z 1132.987,A -85,B 0,C 180,E1 23381.255,E2 23381.255} C_VEL
LIN {X 0,Y 295.671,Z 1150.775,A -85,B 0,C 180,E1 23391.18,E2 23391.18} C_VEL
LIN {X 0,Y 283.176,Z 1160.829,A -85,B 0,C 180,E1 23400.2,E2 23400.2} C_VEL
LIN {X 0,Y 276.32,Z 1164.417,A -85,B 0,C 180,E1 23403.416,E2 23403.416} C_VEL
LIN {X 0,Y 269.856,Z 1167.338,A -85,B 0,C 180,E1 23406.784,E2 23406.784} C_VEL
LIN {X 0,Y 265.059,Z 1170.136,A -85,B 0,C 180,E1 23416.559,E2 23416.559} C_VEL
LIN {X 0,Y 263.588,Z 1169.902,A -85,B 0,C 180,E1 23423.656,E2 23423.656} C_VEL
LIN {X 0,Y 264.341,Z 1166.278,A -85,B 0,C 180,E1 23432.812,E2 23432.812} C_VEL
LIN {X 0,Y 267.117,Z 1160.111,A -85,B 0,C 180,E1 23440.88,E2 23440.88} C_VEL
LIN {X 0,Y 273.184,Z 1148.126,A -85,B 0,C 180,E1 23450.744,E2 23450.744} C_VEL
LIN {X 0,Y 283.698,Z 1131.88,A -85,B 0,C 180,E1 23459.651,E2 23459.651} C_VEL
LIN {X 0,Y 299.236,Z 1108.829,A -85,B 0,C 180,E1 23468.238,E2 23468.238} C_VEL
LIN {X 0,Y 317.294,Z 1082.042,A -85,B 0,C 180,E1 23475.233,E2 23475.233} C_VEL
LIN {X 0,Y 338.58,Z 1047.89,A -85,B 0,C 180,E1 23481.497,E2 23481.497} C_VEL
LIN {X 0,Y 358.807,Z 1011.668,A -85,B 0,C 180,E1 23486.236,E2 23486.236} C_VEL
LIN {X 0,Y 357.359,Z 990.536,A -85,B 0,C 180,E1 23491.464,E2 23491.464} C_VEL
LIN {X 0,Y 353.272,Z 967.862,A -85,B 0,C 180,E1 23497.692,E2 23497.692} C_VEL
LIN {X 0,Y 347.873,Z 949.228,A -85,B 0,C 180,E1 23503.801,E2 23503.801} C_VEL
LIN {X 0,Y 341.842,Z 933.158,A -85,B 0,C 180,E1 23510.206,E2 23510.206} C_VEL
LIN {X 0,Y 335.153,Z 917.978,A -85,B 0,C 180,E1 23518.048,E2 23518.048} C_VEL
LIN {X 0,Y 329.936,Z 907.422,A -85,B 0,C 180,E1 23525.701,E2 23525.701} C_VEL
LIN {X 0,Y 326.451,Z 899.904,A -85,B 0,C 180,E1 23533.987,E2 23533.987} C_VEL
LIN {X 0,Y 324.987,Z 897.503,A -85,B 0,C 180,E1 23542.814,E2 23542.814} C_VEL
LIN {X 0,Y 326.631,Z 898.293,A -85,B 0,C 180,E1 23551.541,E2 23551.541} C_VEL
LIN {X 0,Y 329.195,Z 899.842,A -85,B 0,C 180,E1 23556.666,E2 23556.666} C_VEL
LIN {X 0,Y 334.815,Z 908.04,A -85,B 0,C 180,E1 23564.936,E2 23564.936} C_VEL
LIN {X 0,Y 342.249,Z 919.104,A -85,B 0,C 180,E1 23572.39,E2 23572.39} C_VEL
LIN {X 0,Y 350.004,Z 932.456,A -85,B 0,C 180,E1 23578.686,E2 23578.686} C_VEL
LIN {X 0,Y 359.732,Z 951.196,A -85,B 0,C 180,E1 23585.424,E2 23585.424} C_VEL
LIN {X 0,Y 369.952,Z 973.481,A -85,B 0,C 180,E1 23591.784,E2 23591.784} C_VEL
LIN {X 0,Y 379.695,Z 998.383,A -85,B 0,C 180,E1 23597.665,E2 23597.665} C_VEL
LIN {X 0,Y 385.468,Z 1015.378,A -85,B 0,C 180,E1 23601.201,E2 23601.201} C_VEL
LIN {X 0,Y 365.474,Z 1061.88,A -85,B 0,C 180,E1 23604.529,E2 23604.529} C_VEL
LIN {X 0,Y 343.45,Z 1105.139,A -85,B 0,C 180,E1 23608.944,E2 23608.944} C_VEL
LIN {X 0,Y 322.568,Z 1141.76,A -85,B 0,C 180,E1 23614.203,E2 23614.203} C_VEL
LIN {X 0,Y 301.698,Z 1176.386,A -85,B 0,C 180,E1 23621.282,E2 23621.282} C_VEL
LIN {X 0,Y 284.87,Z 1204.198,A -85,B 0,C 180,E1 23629.459,E2 23629.459} C_VEL
LIN {X 0,Y 273.209,Z 1225.468,A -85,B 0,C 180,E1 23638.314,E2 23638.314} C_VEL
LIN {X 0,Y 267.205,Z 1239.578,A -85,B 0,C 180,E1 23646.667,E2 23646.667} C_VEL
LIN {X 0,Y 264.676,Z 1249.099,A -85,B 0,C 180,E1 23654.989,E2 23654.989} C_VEL
LIN {X 0,Y 264.283,Z 1254.387,A -85,B 0,C 180,E1 23663.42,E2 23663.42} C_VEL
LIN {X 0,Y 265.024,Z 1255.315,A -85,B 0,C 180,E1 23669.987,E2 23669.987} C_VEL
LIN {X 0,Y 264.509,Z 1253.271,A -85,B 0,C 180,E1 23676.547,E2 23676.547} C_VEL
LIN {X 0,Y 265.003,Z 1246.405,A -85,B 0,C 180,E1 23685.15,E2 23685.15} C_VEL
LIN {X 0,Y 267.663,Z 1234.716,A -85,B 0,C 180,E1 23693.942,E2 23693.942} C_VEL
LIN {X 0,Y 274.877,Z 1216.74,A -85,B 0,C 180,E1 23703.332,E2 23703.332} C_VEL
LIN {X 0,Y 289.973,Z 1189.094,A -85,B 0,C 180,E1 23713.649,E2 23713.649} C_VEL
LIN {X 0,Y 316.88,Z 1149.248,A -85,B 0,C 180,E1 23724.14,E2 23724.14} C_VEL
LIN {X 0,Y 348.577,Z 1112.196,A -85,B 0,C 180,E1 23731.521,E2 23731.521} C_VEL
LIN {X 0,Y 309.694,Z 1138.382,A -85,B 0,C 180,E1 23741.509,E2 23741.509} C_VEL
LIN {X 0,Y 288.212,Z 1153.862,A -85,B 0,C 180,E1 23750.95,E2 23750.95} C_VEL
LIN {X 0,Y 274.036,Z 1164.225,A -85,B 0,C 180,E1 23761.579,E2 23761.579} C_VEL
LIN {X 0,Y 269.856,Z 1167.338,A -85,B 0,C 180,E1 23766.784,E2 23766.784} C_VEL
LIN {X 0,Y 263.856,Z 1169.695,A -85,B 0,C 180,E1 23770.273,E2 23770.273} C_VEL
LIN {X 0,Y 258.229,Z 1171.312,A -85,B 0,C 180,E1 23773.907,E2 23773.907} C_VEL
LIN {X 0,Y 256.165,Z 1171.569,A -85,B 0,C 180,E1 23780.725,E2 23780.725} C_VEL
LIN {X 0,Y 255.7,Z 1169.843,A -85,B 0,C 180,E1 23788.211,E2 23788.211} C_VEL
LIN {X 0,Y 257.848,Z 1164.642,A -85,B 0,C 180,E1 23797.211,E2 23797.211} C_VEL
LIN {X 0,Y 262.008,Z 1155.972,A -85,B 0,C 180,E1 23806.225,E2 23806.225} C_VEL
LIN {X 0,Y 271.515,Z 1140.572,A -85,B 0,C 180,E1 23816.588,E2 23816.588} C_VEL
LIN {X 0,Y 286.114,Z 1119.395,A -85,B 0,C 180,E1 23825.864,E2 23825.864} C_VEL
LIN {X 0,Y 304.066,Z 1093.79,A -85,B 0,C 180,E1 23833.619,E2 23833.619} C_VEL
LIN {X 0,Y 325.484,Z 1061.32,A -85,B 0,C 180,E1 23840.436,E2 23840.436} C_VEL
LIN {X 0,Y 346.263,Z 1026.435,A -85,B 0,C 180,E1 23845.578,E2 23845.578} C_VEL
LIN {X 0,Y 352.919,Z 1013.604,A -85,B 0,C 180,E1 23847.193,E2 23847.193} C_VEL
LIN {X 0,Y 351.261,Z 991.578,A -85,B 0,C 180,E1 23852.887,E2 23852.887} C_VEL
LIN {X 0,Y 347.7,Z 971.172,A -85,B 0,C 180,E1 23858.76,E2 23858.76} C_VEL
LIN {X 0,Y 342.182,Z 951.937,A -85,B 0,C 180,E1 23865.375,E2 23865.375} C_VEL
LIN {X 0,Y 336.089,Z 935.448,A -85,B 0,C 180,E1 23872.479,E2 23872.479} C_VEL
LIN {X 0,Y 330.078,Z 921.993,A -85,B 0,C 180,E1 23880.248,E2 23880.248} C_VEL
LIN {X 0,Y 326.134,Z 913.224,A -85,B 0,C 180,E1 23887.05,E2 23887.05} C_VEL
LIN {X 0,Y 323.177,Z 906.667,A -85,B 0,C 180,E1 23895.469,E2 23895.469} C_VEL
LIN {X 0,Y 322.344,Z 904.777,A -85,B 0,C 180,E1 23905.772,E2 23905.772} C_VEL
LIN {X 0,Y 325.699,Z 906.872,A -85,B 0,C 180,E1 23915.322,E2 23915.322} C_VEL
LIN {X 0,Y 331.423,Z 914.217,A -85,B 0,C 180,E1 23924.126,E2 23924.126} C_VEL
LIN {X 0,Y 339.188,Z 926.43,A -85,B 0,C 180,E1 23932.321,E2 23932.321} C_VEL
LIN {X 0,Y 346.941,Z 940.207,A -85,B 0,C 180,E1 23938.754,E2 23938.754} C_VEL
LIN {X 0,Y 357.175,Z 960.811,A -85,B 0,C 180,E1 23946.072,E2 23946.072} C_VEL
LIN {X 0,Y 367.075,Z 983.708,A -85,B 0,C 180,E1 23952.481,E2 23952.481} C_VEL
LIN {X 0,Y 376.814,Z 1010.405,A -85,B 0,C 180,E1 23958.712,E2 23958.712} C_VEL
LIN {X 0,Y 379.256,Z 1018.089,A -85,B 0,C 180,E1 23960.333,E2 23960.333} C_VEL
LIN {X 0,Y 371.179,Z 1038.153,A -85,B 0,C 180,E1 23961.744,E2 23961.744} C_VEL
LIN {X 0,Y 350.397,Z 1081.421,A -85,B 0,C 180,E1 23965.395,E2 23965.395} C_VEL
LIN {X 0,Y 327.27,Z 1123.37,A -85,B 0,C 180,E1 23970.436,E2 23970.436} C_VEL
LIN {X 0,Y 305.282,Z 1159.551,A -85,B 0,C 180,E1 23976.74,E2 23976.74} C_VEL
LIN {X 0,Y 286.602,Z 1189.14,A -85,B 0,C 180,E1 23984.064,E2 23984.064} C_VEL
LIN {X 0,Y 271.157,Z 1214.567,A -85,B 0,C 180,E1 23993.104,E2 23993.104} C_VEL
LIN {X 0,Y 261.781,Z 1232.826,A -85,B 0,C 180,E1 24002.483,E2 24002.483} C_VEL
LIN {X 0,Y 257.66,Z 1244.334,A -85,B 0,C 180,E1 24011.169,E2 24011.169} C_VEL
LIN {X 0,Y 256.474,Z 1251.385,A -85,B 0,C 180,E1 24019.806,E2 24019.806} C_VEL
LIN {X 0,Y 256.749,Z 1253.837,A -85,B 0,C 180,E1 24026.612,E2 24026.612} C_VEL
LIN {X 0,Y 256.987,Z 1253.807,A -85,B 0,C 180,E1 24031.699,E2 24031.699} C_VEL
LIN {X 0,Y 256.657,Z 1249.82,A -85,B 0,C 180,E1 24040.159,E2 24040.159} C_VEL
LIN {X 0,Y 257.877,Z 1241.453,A -85,B 0,C 180,E1 24048.786,E2 24048.786} C_VEL
LIN {X 0,Y 262.449,Z 1227.258,A -85,B 0,C 180,E1 24058.344,E2 24058.344} C_VEL
LIN {X 0,Y 273.346,Z 1205.307,A -85,B 0,C 180,E1 24068.671,E2 24068.671} C_VEL
LIN {X 0,Y 295.746,Z 1170.826,A -85,B 0,C 180,E1 24080.012,E2 24080.012} C_VEL
LIN {X 0,Y 336.602,Z 1122.292,A -85,B 0,C 180,E1 24091.068,E2 24091.068} C_VEL
LIN {X 0,Y 339.456,Z 1119.532,A -85,B 0,C 180,E1 24091.616,E2 24091.616} C_VEL
LIN {X 0,Y 299.196,Z 1144.626,A -85,B 0,C 180,E1 24102.36,E2 24102.36} C_VEL
LIN {X 0,Y 275.796,Z 1160.168,A -85,B 0,C 180,E1 24113.708,E2 24113.708} C_VEL
LIN {X 0,Y 264.736,Z 1167.496,A -85,B 0,C 180,E1 24123.271,E2 24123.271} C_VEL
LIN {X 0,Y 258.229,Z 1171.312,A -85,B 0,C 180,E1 24133.907,E2 24133.907} C_VEL
LIN {X 0,Y 252.983,Z 1172.428,A -85,B 0,C 180,E1 24137.637,E2 24137.637} C_VEL
LIN {X 0,Y 248.209,Z 1172.846,A -85,B 0,C 180,E1 24141.506,E2 24141.506} C_VEL
LIN {X 0,Y 248.779,Z 1168.695,A -85,B 0,C 180,E1 24153.134,E2 24153.134} C_VEL
LIN {X 0,Y 252.029,Z 1161.806,A -85,B 0,C 180,E1 24162.182,E2 24162.182} C_VEL
LIN {X 0,Y 259.404,Z 1148.918,A -85,B 0,C 180,E1 24172.886,E2 24172.886} C_VEL
LIN {X 0,Y 271.428,Z 1131.538,A -85,B 0,C 180,E1 24182.231,E2 24182.231} C_VEL
LIN {X 0,Y 288.101,Z 1108.559,A -85,B 0,C 180,E1 24190.738,E2 24190.738} C_VEL
LIN {X 0,Y 307.178,Z 1081.518,A -85,B 0,C 180,E1 24197.674,E2 24197.674} C_VEL
LIN {X 0,Y 329.372,Z 1047.443,A -85,B 0,C 180,E1 24203.832,E2 24203.832} C_VEL
LIN {X 0,Y 346.891,Z 1017.205,A -85,B 0,C 180,E1 24207.826,E2 24207.826} C_VEL
LIN {X 0,Y 345.622,Z 996.313,A -85,B 0,C 180,E1 24213.353,E2 24213.353} C_VEL
LIN {X 0,Y 342.371,Z 975.574,A -85,B 0,C 180,E1 24219.537,E2 24219.537} C_VEL
LIN {X 0,Y 337.101,Z 956.503,A -85,B 0,C 180,E1 24226.334,E2 24226.334} C_VEL
LIN {X 0,Y 331.722,Z 941.434,A -85,B 0,C 180,E1 24233.06,E2 24233.06} C_VEL
LIN {X 0,Y 326.339,Z 928.604,A -85,B 0,C 180,E1 24240.632,E2 24240.632} C_VEL
LIN {X 0,Y 322.771,Z 920.124,A -85,B 0,C 180,E1 24247.501,E2 24247.501} C_VEL
LIN {X 0,Y 320.249,Z 914.137,A -85,B 0,C 180,E1 24255.068,E2 24255.068} C_VEL
LIN {X 0,Y 319.328,Z 912.204,A -85,B 0,C 180,E1 24263.574,E2 24263.574} C_VEL
LIN {X 0,Y 321.156,Z 913.163,A -85,B 0,C 180,E1 24271.935,E2 24271.935} C_VEL
LIN {X 0,Y 324.257,Z 916.185,A -85,B 0,C 180,E1 24278.113,E2 24278.113} C_VEL
LIN {X 0,Y 328.892,Z 922.801,A -85,B 0,C 180,E1 24284.796,E2 24284.796} C_VEL
LIN {X 0,Y 336.116,Z 933.784,A -85,B 0,C 180,E1 24292.25,E2 24292.25} C_VEL
LIN {X 0,Y 343.658,Z 947.832,A -85,B 0,C 180,E1 24298.837,E2 24298.837} C_VEL
LIN {X 0,Y 353.221,Z 967.786,A -85,B 0,C 180,E1 24305.941,E2 24305.941} C_VEL
LIN {X 0,Y 362.577,Z 990.342,A -85,B 0,C 180,E1 24312.333,E2 24312.333} C_VEL
LIN {X 0,Y 371.478,Z 1015.804,A -85,B 0,C 180,E1 24318.376,E2 24318.376} C_VEL
LIN {X 0,Y 373.368,Z 1021.887,A -85,B 0,C 180,E1 24319.679,E2 24319.679} C_VEL
LIN {X 0,Y 352.904,Z 1066.283,A -85,B 0,C 180,E1 24323.014,E2 24323.014} C_VEL
LIN {X 0,Y 330.661,Z 1107.511,A -85,B 0,C 180,E1 24327.37,E2 24327.37} C_VEL
LIN {X 0,Y 307.28,Z 1146.015,A -85,B 0,C 180,E1 24333.262,E2 24333.262} C_VEL
LIN {X 0,Y 286.911,Z 1177.625,A -85,B 0,C 180,E1 24340.193,E2 24340.193} C_VEL
LIN {X 0,Y 268.828,Z 1205.584,A -85,B 0,C 180,E1 24349.065,E2 24349.065} C_VEL
LIN {X 0,Y 257.341,Z 1225.164,A -85,B 0,C 180,E1 24358.082,E2 24358.082} C_VEL
LIN {X 0,Y 250.892,Z 1239.759,A -85,B 0,C 180,E1 24367.873,E2 24367.873} C_VEL
LIN {X 0,Y 248.891,Z 1247.867,A -85,B 0,C 180,E1 24376.255,E2 24376.255} C_VEL
LIN {X 0,Y 248.644,Z 1251.642,A -85,B 0,C 180,E1 24383.005,E2 24383.005} C_VEL
LIN {X 0,Y 249.448,Z 1252.628,A -85,B 0,C 180,E1 24389.986,E2 24389.986} C_VEL
LIN {X 0,Y 248.86,Z 1250.62,A -85,B 0,C 180,E1 24396.961,E2 24396.961} C_VEL
LIN {X 0,Y 249.387,Z 1244.027,A -85,B 0,C 180,E1 24405.808,E2 24405.808} C_VEL
LIN {X 0,Y 252.692,Z 1231.815,A -85,B 0,C 180,E1 24415.617,E2 24415.617} C_VEL
LIN {X 0,Y 262.477,Z 1211.422,A -85,B 0,C 180,E1 24426.649,E2 24426.649} C_VEL
LIN {X 0,Y 282.071,Z 1181.477,A -85,B 0,C 180,E1 24437.967,E2 24437.967} C_VEL
LIN {X 0,Y 326.139,Z 1130.387,A -85,B 0,C 180,E1 24450.955,E2 24450.955} C_VEL
LIN {X 0,Y 329.886,Z 1126.66,A -85,B 0,C 180,E1 24451.772,E2 24451.772} C_VEL
LIN {X 0,Y 290.395,Z 1149.366,A -85,B 0,C 180,E1 24462.59,E2 24462.59} C_VEL
LIN {X 0,Y 268.158,Z 1162.844,A -85,B 0,C 180,E1 24473.528,E2 24473.528} C_VEL
LIN {X 0,Y 256.853,Z 1169.667,A -85,B 0,C 180,E1 24483.371,E2 24483.371} C_VEL
LIN {X 0,Y 250.451,Z 1172.995,A -85,B 0,C 180,E1 24493.963,E2 24493.963} C_VEL
LIN {X 0,Y 248.209,Z 1172.846,A -85,B 0,C 180,E1 24501.506,E2 24501.506} C_VEL
LIN {X 0,Y 243.855,Z 1172.66,A -85,B 0,C 180,E1 24505.46,E2 24505.46} C_VEL
LIN {X 0,Y 240.203,Z 1171.808,A -85,B 0,C 180,E1 24509.534,E2 24509.534} C_VEL
LIN {X 0,Y 243.119,Z 1165.448,A -85,B 0,C 180,E1 24519.725,E2 24519.725} C_VEL
LIN {X 0,Y 248.535,Z 1155.529,A -85,B 0,C 180,E1 24529.506,E2 24529.506} C_VEL
LIN {X 0,Y 259.641,Z 1139.242,A -85,B 0,C 180,E1 24539.831,E2 24539.831} C_VEL
LIN {X 0,Y 275.406,Z 1118.183,A -85,B 0,C 180,E1 24548.854,E2 24548.854} C_VEL
LIN {X 0,Y 295.498,Z 1090.702,A -85,B 0,C 180,E1 24556.805,E2 24556.805} C_VEL
LIN {X 0,Y 316.648,Z 1059.97,A -85,B 0,C 180,E1 24563.018,E2 24563.018} C_VEL
LIN {X 0,Y 340.085,Z 1021.637,A -85,B 0,C 180,E1 24568.419,E2 24568.419} C_VEL
LIN {X 0,Y 340.709,Z 1014.956,A -85,B 0,C 180,E1 24570.01,E2 24570.01} C_VEL
LIN {X 0,Y 339.266,Z 994.439,A -85,B 0,C 180,E1 24575.762,E2 24575.762} C_VEL
LIN {X 0,Y 336.431,Z 977.448,A -85,B 0,C 180,E1 24581.161,E2 24581.161} C_VEL
LIN {X 0,Y 331.562,Z 959.457,A -85,B 0,C 180,E1 24587.982,E2 24587.982} C_VEL
LIN {X 0,Y 326.681,Z 945.69,A -85,B 0,C 180,E1 24594.612,E2 24594.612} C_VEL
LIN {X 0,Y 321.907,Z 933.298,A -85,B 0,C 180,E1 24602.341,E2 24602.341} C_VEL
LIN {X 0,Y 318.644,Z 925.792,A -85,B 0,C 180,E1 24609.332,E2 24609.332} C_VEL
LIN {X 0,Y 316.953,Z 921.209,A -85,B 0,C 180,E1 24615.668,E2 24615.668} C_VEL
LIN {X 0,Y 316.412,Z 919.451,A -85,B 0,C 180,E1 24625.038,E2 24625.038} C_VEL
LIN {X 0,Y 319.686,Z 921.429,A -85,B 0,C 180,E1 24634.826,E2 24634.826} C_VEL
LIN {X 0,Y 325.31,Z 928.73,A -85,B 0,C 180,E1 24643.819,E2 24643.819} C_VEL
LIN {X 0,Y 332.753,Z 940.972,A -85,B 0,C 180,E1 24652.171,E2 24652.171} C_VEL
LIN {X 0,Y 340.146,Z 954.994,A -85,B 0,C 180,E1 24658.728,E2 24658.728} C_VEL
LIN {X 0,Y 348.78,Z 973.726,A -85,B 0,C 180,E1 24665.494,E2 24665.494} C_VEL
LIN {X 0,Y 357.583,Z 995.807,A -85,B 0,C 180,E1 24671.889,E2 24671.889} C_VEL
LIN {X 0,Y 366.17,Z 1021.186,A -85,B 0,C 180,E1 24678.03,E2 24678.03} C_VEL
LIN {X 0,Y 366.995,Z 1026.075,A -85,B 0,C 180,E1 24678.972,E2 24678.972} C_VEL
LIN {X 0,Y 343.971,Z 1073.469,A -85,B 0,C 180,E1 24682.677,E2 24682.677} C_VEL
LIN {X 0,Y 321.334,Z 1113.571,A -85,B 0,C 180,E1 24687.225,E2 24687.225} C_VEL
LIN {X 0,Y 299.262,Z 1148.791,A -85,B 0,C 180,E1 24692.886,E2 24692.886} C_VEL
LIN {X 0,Y 277.712,Z 1180.848,A -85,B 0,C 180,E1 24700.362,E2 24700.362} C_VEL
LIN {X 0,Y 260.753,Z 1206.248,A -85,B 0,C 180,E1 24708.88,E2 24708.88} C_VEL
LIN {X 0,Y 248.696,Z 1226.223,A -85,B 0,C 180,E1 24718.708,E2 24718.708} C_VEL
LIN {X 0,Y 242.608,Z 1240.469,A -85,B 0,C 180,E1 24729.106,E2 24729.106} C_VEL
LIN {X 0,Y 240.935,Z 1247.698,A -85,B 0,C 180,E1 24737.681,E2 24737.681} C_VEL
LIN {X 0,Y 241.141,Z 1251.084,A -85,B 0,C 180,E1 24746.393,E2 24746.393} C_VEL
LIN {X 0,Y 241.671,Z 1251.29,A -85,B 0,C 180,E1 24749.985,E2 24749.985} C_VEL
LIN {X 0,Y 241.058,Z 1249.296,A -85,B 0,C 180,E1 24757.187,E2 24757.187} C_VEL
LIN {X 0,Y 241.601,Z 1242.647,A -85,B 0,C 180,E1 24766.331,E2 24766.331} C_VEL
LIN {X 0,Y 245.229,Z 1230.472,A -85,B 0,C 180,E1 24776.456,E2 24776.456} C_VEL
LIN {X 0,Y 255.677,Z 1210.41,A -85,B 0,C 180,E1 24787.718,E2 24787.718} C_VEL
LIN {X 0,Y 278.37,Z 1178.497,A -85,B 0,C 180,E1 24800.029,E2 24800.029} C_VEL
LIN {X 0,Y 320.56,Z 1133.312,A -85,B 0,C 180,E1 24811.876,E2 24811.876} C_VEL
LIN {X 0,Y 281.592,Z 1153.988,A -85,B 0,C 180,E1 24822.834,E2 24822.834} C_VEL
LIN {X 0,Y 257.637,Z 1167.263,A -85,B 0,C 180,E1 24835.424,E2 24835.424} C_VEL
LIN {X 0,Y 246.32,Z 1173.104,A -85,B 0,C 180,E1 24847.046,E2 24847.046} C_VEL
LIN {X 0,Y 241.141,Z 1174.644,A -85,B 0,C 180,E1 24858.257,E2 24858.257} C_VEL
LIN {X 0,Y 240.203,Z 1171.808,A -85,B 0,C 180,E1 24869.534,E2 24869.534} C_VEL
LIN {X 0,Y 238.333,Z 1170.749,A -85,B 0,C 180,E1 24872.63,E2 24872.63} C_VEL
LIN {X 0,Y 234.568,Z 1168.271,A -85,B 0,C 180,E1 24877.86,E2 24877.86} C_VEL
LIN {X 0,Y 239.124,Z 1159.774,A -85,B 0,C 180,E1 24887.282,E2 24887.282} C_VEL
LIN {X 0,Y 249.221,Z 1144.918,A -85,B 0,C 180,E1 24898.079,E2 24898.079} C_VEL
LIN {X 0,Y 264.149,Z 1125.312,A -85,B 0,C 180,E1 24907.45,E2 24907.45} C_VEL
LIN {X 0,Y 284.857,Z 1098.357,A -85,B 0,C 180,E1 24916.165,E2 24916.165} C_VEL
LIN {X 0,Y 307.946,Z 1065.874,A -85,B 0,C 180,E1 24923.203,E2 24923.203} C_VEL
LIN {X 0,Y 330.194,Z 1031.139,A -85,B 0,C 180,E1 24928.415,E2 24928.415} C_VEL
LIN {X 0,Y 334.774,Z 1023.023,A -85,B 0,C 180,E1 24929.461,E2 24929.461} C_VEL
LIN {X 0,Y 333.946,Z 1001.778,A -85,B 0,C 180,E1 24935.495,E2 24935.495} C_VEL
LIN {X 0,Y 331.506,Z 984.004,A -85,B 0,C 180,E1 24941.181,E2 24941.181} C_VEL
LIN {X 0,Y 327.134,Z 965.945,A -85,B 0,C 180,E1 24948.18,E2 24948.18} C_VEL
LIN {X 0,Y 322.631,Z 952.183,A -85,B 0,C 180,E1 24954.942,E2 24954.942} C_VEL
LIN {X 0,Y 318.176,Z 939.936,A -85,B 0,C 180,E1 24962.768,E2 24962.768} C_VEL
LIN {X 0,Y 315.043,Z 932.485,A -85,B 0,C 180,E1 24969.882,E2 24969.882} C_VEL
LIN {X 0,Y 313.648,Z 928.239,A -85,B 0,C 180,E1 24976.29,E2 24976.29} C_VEL
LIN {X 0,Y 313.294,Z 926.692,A -85,B 0,C 180,E1 24985.097,E2 24985.097} C_VEL
LIN {X 0,Y 316.676,Z 928.862,A -85,B 0,C 180,E1 24995.066,E2 24995.066} C_VEL
LIN {X 0,Y 321.967,Z 935.847,A -85,B 0,C 180,E1 25003.647,E2 25003.647} C_VEL
LIN {X 0,Y 329.372,Z 948.185,A -85,B 0,C 180,E1 25012.091,E2 25012.091} C_VEL
LIN {X 0,Y 336.654,Z 962.575,A -85,B 0,C 180,E1 25018.841,E2 25018.841} C_VEL
LIN {X 0,Y 344.99,Z 981.287,A -85,B 0,C 180,E1 25025.583,E2 25025.583} C_VEL
LIN {X 0,Y 353.838,Z 1004.539,A -85,B 0,C 180,E1 25032.329,E2 25032.329} C_VEL
LIN {X 0,Y 361.171,Z 1027.893,A -85,B 0,C 180,E1 25038.011,E2 25038.011} C_VEL
LIN {X 0,Y 338.612,Z 1073.901,A -85,B 0,C 180,E1 25041.709,E2 25041.709} C_VEL
LIN {X 0,Y 314.704,Z 1114.953,A -85,B 0,C 180,E1 25046.436,E2 25046.436} C_VEL
LIN {X 0,Y 292.304,Z 1149.611,A -85,B 0,C 180,E1 25052.145,E2 25052.145} C_VEL
LIN {X 0,Y 270.06,Z 1181.685,A -85,B 0,C 180,E1 25059.853,E2 25059.853} C_VEL
LIN {X 0,Y 253.47,Z 1205.676,A -85,B 0,C 180,E1 25068.22,E2 25068.22} C_VEL
LIN {X 0,Y 240.9,Z 1225.753,A -85,B 0,C 180,E1 25078.459,E2 25078.459} C_VEL
LIN {X 0,Y 234.879,Z 1239.223,A -85,B 0,C 180,E1 25088.692,E2 25088.692} C_VEL
LIN {X 0,Y 233.04,Z 1247.176,A -85,B 0,C 180,E1 25098.768,E2 25098.768} C_VEL
LIN {X 0,Y 233.348,Z 1249.715,A -85,B 0,C 180,E1 25106.272,E2 25106.272} C_VEL
LIN {X 0,Y 233.897,Z 1249.937,A -85,B 0,C 180,E1 25109.985,E2 25109.985} C_VEL
LIN {X 0,Y 233.229,Z 1247.934,A -85,B 0,C 180,E1 25117.43,E2 25117.43} C_VEL
LIN {X 0,Y 233.829,Z 1241.279,A -85,B 0,C 180,E1 25126.89,E2 25126.89} C_VEL
LIN {X 0,Y 237.999,Z 1228.718,A -85,B 0,C 180,E1 25137.657,E2 25137.657} C_VEL
LIN {X 0,Y 249.717,Z 1208.235,A -85,B 0,C 180,E1 25149.428,E2 25149.428} C_VEL
LIN {X 0,Y 275.111,Z 1175.634,A -85,B 0,C 180,E1 25162.185,E2 25162.185} C_VEL
LIN {X 0,Y 310.552,Z 1140.056,A -85,B 0,C 180,E1 25172.12,E2 25172.12} C_VEL
LIN {X 0,Y 270.959,Z 1159.223,A -85,B 0,C 180,E1 25183.809,E2 25183.809} C_VEL
LIN {X 0,Y 249.933,Z 1169.735,A -85,B 0,C 180,E1 25195.283,E2 25195.283} C_VEL
LIN {X 0,Y 238.363,Z 1175.06,A -85,B 0,C 180,E1 25207.282,E2 25207.282} C_VEL
LIN {X 0,Y 233.139,Z 1175.928,A -85,B 0,C 180,E1 25218.907,E2 25218.907} C_VEL
LIN {X 0,Y 232.364,Z 1173.055,A -85,B 0,C 180,E1 25229.634,E2 25229.634} C_VEL
LIN {X 0,Y 234.568,Z 1168.271,A -85,B 0,C 180,E1 25237.86,E2 25237.86} C_VEL
LIN {X 0,Y 233.304,Z 1166.34,A -85,B 0,C 180,E1 25241.028,E2 25241.028} C_VEL
LIN {X 0,Y 230.466,Z 1163.029,A -85,B 0,C 180,E1 25245.833,E2 25245.833} C_VEL
LIN {X 0,Y 230.685,Z 1162.482,A -85,B 0,C 180,E1 25246.362,E2 25246.362} C_VEL
LIN {X 0,Y 240.794,Z 1147.63,A -85,B 0,C 180,E1 25257.821,E2 25257.821} C_VEL
LIN {X 0,Y 255.922,Z 1128.526,A -85,B 0,C 180,E1 25267.537,E2 25267.537} C_VEL
LIN {X 0,Y 276.252,Z 1102.726,A -85,B 0,C 180,E1 25276.269,E2 25276.269} C_VEL
LIN {X 0,Y 297.564,Z 1073.992,A -85,B 0,C 180,E1 25282.949,E2 25282.949} C_VEL
LIN {X 0,Y 322.337,Z 1036.934,A -85,B 0,C 180,E1 25288.87,E2 25288.87} C_VEL
LIN {X 0,Y 328.724,Z 1026.164,A -85,B 0,C 180,E1 25290.245,E2 25290.245} C_VEL
LIN {X 0,Y 328.284,Z 1005.641,A -85,B 0,C 180,E1 25296.287,E2 25296.287} C_VEL
LIN {X 0,Y 326.012,Z 987.811,A -85,B 0,C 180,E1 25302.211,E2 25302.211} C_VEL
LIN {X 0,Y 322.282,Z 971.499,A -85,B 0,C 180,E1 25308.736,E2 25308.736} C_VEL
LIN {X 0,Y 317.822,Z 956.969,A -85,B 0,C 180,E1 25316.138,E2 25316.138} C_VEL
LIN {X 0,Y 314.175,Z 946.334,A -85,B 0,C 180,E1 25323.304,E2 25323.304} C_VEL
LIN {X 0,Y 311.856,Z 940.221,A -85,B 0,C 180,E1 25329.176,E2 25329.176} C_VEL
LIN {X 0,Y 310.139,Z 935.178,A -85,B 0,C 180,E1 25336.995,E2 25336.995} C_VEL
LIN {X 0,Y 310.277,Z 934.004,A -85,B 0,C 180,E1 25345.904,E2 25345.904} C_VEL
LIN {X 0,Y 313.076,Z 935.733,A -85,B 0,C 180,E1 25354.256,E2 25354.256} C_VEL
LIN {X 0,Y 317.538,Z 941.85,A -85,B 0,C 180,E1 25362.16,E2 25362.16} C_VEL
LIN {X 0,Y 323.974,Z 952.252,A -85,B 0,C 180,E1 25370.071,E2 25370.071} C_VEL
LIN {X 0,Y 329.931,Z 963.32,A -85,B 0,C 180,E1 25376.061,E2 25376.061} C_VEL
LIN {X 0,Y 337.999,Z 981.35,A -85,B 0,C 180,E1 25383.204,E2 25383.204} C_VEL
LIN {X 0,Y 346.426,Z 1003.232,A -85,B 0,C 180,E1 25390.049,E2 25390.049} C_VEL
LIN {X 0,Y 354.115,Z 1027.829,A -85,B 0,C 180,E1 25396.421,E2 25396.421} C_VEL
LIN {X 0,Y 354.532,Z 1032.857,A -85,B 0,C 180,E1 25397.39,E2 25397.39} C_VEL
LIN {X 0,Y 332.061,Z 1076.49,A -85,B 0,C 180,E1 25400.927,E2 25400.927} C_VEL
LIN {X 0,Y 306.702,Z 1118.625,A -85,B 0,C 180,E1 25405.929,E2 25405.929} C_VEL
LIN {X 0,Y 282.745,Z 1153.991,A -85,B 0,C 180,E1 25412.128,E2 25412.128} C_VEL
LIN {X 0,Y 261.736,Z 1183.503,A -85,B 0,C 180,E1 25419.632,E2 25419.632} C_VEL
LIN {X 0,Y 243.416,Z 1209.054,A -85,B 0,C 180,E1 25429.303,E2 25429.303} C_VEL
LIN {X 0,Y 231.951,Z 1227.493,A -85,B 0,C 180,E1 25439.659,E2 25439.659} C_VEL
LIN {X 0,Y 226.463,Z 1239.991,A -85,B 0,C 180,E1 25450.495,E2 25450.495} C_VEL
LIN {X 0,Y 225.239,Z 1245.726,A -85,B 0,C 180,E1 25458.373,E2 25458.373} C_VEL
LIN {X 0,Y 225.525,Z 1248.31,A -85,B 0,C 180,E1 25466.143,E2 25466.143} C_VEL
LIN {X 0,Y 226.101,Z 1248.59,A -85,B 0,C 180,E1 25469.984,E2 25469.984} C_VEL
LIN {X 0,Y 225.404,Z 1246.562,A -85,B 0,C 180,E1 25477.689,E2 25477.689} C_VEL
LIN {X 0,Y 226.079,Z 1239.913,A -85,B 0,C 180,E1 25487.487,E2 25487.487} C_VEL
LIN {X 0,Y 230.269,Z 1228.151,A -85,B 0,C 180,E1 25498.05,E2 25498.05} C_VEL
LIN {X 0,Y 241.945,Z 1209.064,A -85,B 0,C 180,E1 25509.784,E2 25509.784} C_VEL
LIN {X 0,Y 268.254,Z 1177.178,A -85,B 0,C 180,E1 25522.968,E2 25522.968} C_VEL
LIN {X 0,Y 299.366,Z 1147.612,A -85,B 0,C 180,E1 25531.685,E2 25531.685} C_VEL
LIN {X 0,Y 300.628,Z 1146.213,A -85,B 0,C 180,E1 25532.311,E2 25532.311} C_VEL
LIN {X 0,Y 260.619,Z 1164.093,A -85,B 0,C 180,E1 25544.722,E2 25544.722} C_VEL
LIN {X 0,Y 240.583,Z 1172.936,A -85,B 0,C 180,E1 25556.398,E2 25556.398} C_VEL
LIN {X 0,Y 229.425,Z 1177.14,A -85,B 0,C 180,E1 25569.008,E2 25569.008} C_VEL
LIN {X 0,Y 225.041,Z 1177.165,A -85,B 0,C 180,E1 25579.989,E2 25579.989} C_VEL
LIN {X 0,Y 225.155,Z 1173.007,A -85,B 0,C 180,E1 25592.469,E2 25592.469} C_VEL
LIN {X 0,Y 228.192,Z 1166.985,A -85,B 0,C 180,E1 25601.463,E2 25601.463} C_VEL
LIN {X 0,Y 230.685,Z 1162.482,A -85,B 0,C 180,E1 25606.362,E2 25606.362} C_VEL
LIN {X 0,Y 229.634,Z 1158.703,A -85,B 0,C 180,E1 25610.603,E2 25610.603} C_VEL
LIN {X 0,Y 229.439,Z 1154.241,A -85,B 0,C 180,E1 25614.861,E2 25614.861} C_VEL
LIN {X 0,Y 243.642,Z 1136.372,A -85,B 0,C 180,E1 25625.403,E2 25625.403} C_VEL
LIN {X 0,Y 264.03,Z 1111.608,A -85,B 0,C 180,E1 25635.029,E2 25635.029} C_VEL
LIN {X 0,Y 287.316,Z 1081.517,A -85,B 0,C 180,E1 25642.71,E2 25642.71} C_VEL
LIN {X 0,Y 310.563,Z 1048.613,A -85,B 0,C 180,E1 25648.473,E2 25648.473} C_VEL
LIN {X 0,Y 322.571,Z 1029.624,A -85,B 0,C 180,E1 25651.018,E2 25651.018} C_VEL
LIN {X 0,Y 322.757,Z 1011.962,A -85,B 0,C 180,E1 25656.292,E2 25656.292} C_VEL
LIN {X 0,Y 320.955,Z 993.901,A -85,B 0,C 180,E1 25662.406,E2 25662.406} C_VEL
LIN {X 0,Y 317.884,Z 978.677,A -85,B 0,C 180,E1 25668.564,E2 25668.564} C_VEL
LIN {X 0,Y 313.942,Z 964.726,A -85,B 0,C 180,E1 25675.682,E2 25675.682} C_VEL
LIN {X 0,Y 310.499,Z 953.688,A -85,B 0,C 180,E1 25683.092,E2 25683.092} C_VEL
LIN {X 0,Y 307.866,Z 946.114,A -85,B 0,C 180,E1 25690.778,E2 25690.778} C_VEL
LIN {X 0,Y 306.626,Z 942.158,A -85,B 0,C 180,E1 25697.68,E2 25697.68} C_VEL
LIN {X 0,Y 307.247,Z 941.299,A -85,B 0,C 180,E1 25707.252,E2 25707.252} C_VEL
LIN {X 0,Y 309.658,Z 942.842,A -85,B 0,C 180,E1 25713.951,E2 25713.951} C_VEL
LIN {X 0,Y 312.836,Z 947.474,A -85,B 0,C 180,E1 25720.24,E2 25720.24} C_VEL
LIN {X 0,Y 316.371,Z 952.691,A -85,B 0,C 180,E1 25725.284,E2 25725.284} C_VEL
LIN {X 0,Y 322.183,Z 962.364,A -85,B 0,C 180,E1 25731.913,E2 25731.913} C_VEL
LIN {X 0,Y 328.777,Z 976.285,A -85,B 0,C 180,E1 25738.5,E2 25738.5} C_VEL
LIN {X 0,Y 336.122,Z 994.251,A -85,B 0,C 180,E1 25745.159,E2 25745.159} C_VEL
LIN {X 0,Y 344.145,Z 1017.365,A -85,B 0,C 180,E1 25752.038,E2 25752.038} C_VEL
LIN {X 0,Y 348.932,Z 1034.214,A -85,B 0,C 180,E1 25756.35,E2 25756.35} C_VEL
LIN {X 0,Y 327.914,Z 1074.823,A -85,B 0,C 180,E1 25759.718,E2 25759.718} C_VEL
LIN {X 0,Y 301.581,Z 1117.754,A -85,B 0,C 180,E1 25764.773,E2 25764.773} C_VEL
LIN {X 0,Y 276.753,Z 1153.454,A -85,B 0,C 180,E1 25771.062,E2 25771.062} C_VEL
LIN {X 0,Y 254.59,Z 1183.478,A -85,B 0,C 180,E1 25778.879,E2 25778.879} C_VEL
LIN {X 0,Y 235.674,Z 1209.056,A -85,B 0,C 180,E1 25788.904,E2 25788.904} C_VEL
LIN {X 0,Y 224.01,Z 1227.104,A -85,B 0,C 180,E1 25799.59,E2 25799.59} C_VEL
LIN {X 0,Y 218.812,Z 1238.441,A -85,B 0,C 180,E1 25809.784,E2 25809.784} C_VEL
LIN {X 0,Y 217.459,Z 1244.234,A -85,B 0,C 180,E1 25817.951,E2 25817.951} C_VEL
LIN {X 0,Y 217.702,Z 1246.928,A -85,B 0,C 180,E1 25826.004,E2 25826.004} C_VEL
LIN {X 0,Y 218.324,Z 1247.234,A -85,B 0,C 180,E1 25829.984,E2 25829.984} C_VEL
LIN {X 0,Y 217.572,Z 1245.192,A -85,B 0,C 180,E1 25837.968,E2 25837.968} C_VEL
LIN {X 0,Y 218.025,Z 1240.252,A -85,B 0,C 180,E1 25846.078,E2 25846.078} C_VEL
LIN {X 0,Y 222.19,Z 1228.392,A -85,B 0,C 180,E1 25857.861,E2 25857.861} C_VEL
LIN {X 0,Y 234.167,Z 1209.693,A -85,B 0,C 180,E1 25870.167,E2 25870.167} C_VEL
LIN {X 0,Y 260.555,Z 1179.753,A -85,B 0,C 180,E1 25883.464,E2 25883.464} C_VEL
LIN {X 0,Y 291.666,Z 1151.918,A -85,B 0,C 180,E1 25892.208,E2 25892.208} C_VEL
LIN {X 0,Y 249.619,Z 1168.719,A -85,B 0,C 180,E1 25905.987,E2 25905.987} C_VEL
LIN {X 0,Y 228.657,Z 1176.83,A -85,B 0,C 180,E1 25919.999,E2 25919.999} C_VEL
LIN {X 0,Y 220.12,Z 1179.104,A -85,B 0,C 180,E1 25931.882,E2 25931.882} C_VEL
LIN {X 0,Y 217.177,Z 1178.49,A -85,B 0,C 180,E1 25940.355,E2 25940.355} C_VEL
LIN {X 0,Y 217.072,Z 1174.874,A -85,B 0,C 180,E1 25951.386,E2 25951.386} C_VEL
LIN {X 0,Y 220.103,Z 1168.763,A -85,B 0,C 180,E1 25960.984,E2 25960.984} C_VEL
LIN {X 0,Y 226.201,Z 1158.839,A -85,B 0,C 180,E1 25971.297,E2 25971.297} C_VEL
LIN {X 0,Y 229.439,Z 1154.241,A -85,B 0,C 180,E1 25974.861,E2 25974.861} C_VEL
LIN {X 0,Y 230.124,Z 1149.259,A -85,B 0,C 180,E1 25979.054,E2 25979.054} C_VEL
LIN {X 0,Y 231.693,Z 1143.527,A -85,B 0,C 180,E1 25983.16,E2 25983.16} C_VEL
LIN {X 0,Y 250.455,Z 1121.479,A -85,B 0,C 180,E1 25993.117,E2 25993.117} C_VEL
LIN {X 0,Y 273.967,Z 1092.779,A -85,B 0,C 180,E1 26001.553,E2 26001.553} C_VEL
LIN {X 0,Y 297.465,Z 1061.266,A -85,B 0,C 180,E1 26007.808,E2 26007.808} C_VEL
LIN {X 0,Y 316.798,Z 1031.822,A -85,B 0,C 180,E1 26012.072,E2 26012.072} C_VEL
LIN {X 0,Y 316.907,Z 1012.252,A -85,B 0,C 180,E1 26018.235,E2 26018.235} C_VEL
LIN {X 0,Y 315.209,Z 995.955,A -85,B 0,C 180,E1 26024.143,E2 26024.143} C_VEL
LIN {X 0,Y 312.071,Z 980.129,A -85,B 0,C 180,E1 26031.042,E2 26031.042} C_VEL
LIN {X 0,Y 308.592,Z 967.587,A -85,B 0,C 180,E1 26038.197,E2 26038.197} C_VEL
LIN {X 0,Y 306.08,Z 958.942,A -85,B 0,C 180,E1 26044.566,E2 26044.566} C_VEL
LIN {X 0,Y 303.931,Z 952.356,A -85,B 0,C 180,E1 26051.781,E2 26051.781} C_VEL
LIN {X 0,Y 303.068,Z 948.865,A -85,B 0,C 180,E1 26059.6,E2 26059.6} C_VEL
LIN {X 0,Y 303.91,Z 948.497,A -85,B 0,C 180,E1 26067.72,E2 26067.72} C_VEL
LIN {X 0,Y 306.062,Z 949.834,A -85,B 0,C 180,E1 26073.621,E2 26073.621} C_VEL
LIN {X 0,Y 309.231,Z 954.4,A -85,B 0,C 180,E1 26080,E2 26080} C_VEL
LIN {X 0,Y 312.747,Z 959.629,A -85,B 0,C 180,E1 26085.128,E2 26085.128} C_VEL
LIN {X 0,Y 318.934,Z 970.291,A -85,B 0,C 180,E1 26092.308,E2 26092.308} C_VEL
LIN {X 0,Y 325.609,Z 985.424,A -85,B 0,C 180,E1 26099.336,E2 26099.336} C_VEL
LIN {X 0,Y 332.899,Z 1004.392,A -85,B 0,C 180,E1 26106.189,E2 26106.189} C_VEL
LIN {X 0,Y 340.103,Z 1027.06,A -85,B 0,C 180,E1 26112.836,E2 26112.836} C_VEL
LIN {X 0,Y 342.581,Z 1038.838,A -85,B 0,C 180,E1 26115.675,E2 26115.675} C_VEL
LIN {X 0,Y 316.572,Z 1085.548,A -85,B 0,C 180,E1 26119.726,E2 26119.726} C_VEL
LIN {X 0,Y 292.411,Z 1122.793,A -85,B 0,C 180,E1 26124.485,E2 26124.485} C_VEL
LIN {X 0,Y 266.765,Z 1158.393,A -85,B 0,C 180,E1 26131.168,E2 26131.168} C_VEL
LIN {X 0,Y 243.534,Z 1188.533,A -85,B 0,C 180,E1 26139.818,E2 26139.818} C_VEL
LIN {X 0,Y 226.935,Z 1210.41,A -85,B 0,C 180,E1 26149.191,E2 26149.191} C_VEL
LIN {X 0,Y 215.315,Z 1227.951,A -85,B 0,C 180,E1 26160.559,E2 26160.559} C_VEL
LIN {X 0,Y 210.587,Z 1238.561,A -85,B 0,C 180,E1 26171.144,E2 26171.144} C_VEL
LIN {X 0,Y 209.671,Z 1242.717,A -85,B 0,C 180,E1 26177.497,E2 26177.497} C_VEL
LIN {X 0,Y 209.902,Z 1245.515,A -85,B 0,C 180,E1 26185.855,E2 26185.855} C_VEL
LIN {X 0,Y 210.538,Z 1245.886,A -85,B 0,C 180,E1 26189.983,E2 26189.983} C_VEL
LIN {X 0,Y 209.747,Z 1243.821,A -85,B 0,C 180,E1 26198.267,E2 26198.267} C_VEL
LIN {X 0,Y 210.246,Z 1238.934,A -85,B 0,C 180,E1 26206.69,E2 26206.69} C_VEL
LIN {X 0,Y 214.675,Z 1227.459,A -85,B 0,C 180,E1 26218.652,E2 26218.652} C_VEL
LIN {X 0,Y 228.693,Z 1207.534,A -85,B 0,C 180,E1 26232.211,E2 26232.211} C_VEL
LIN {X 0,Y 260.366,Z 1175.274,A -85,B 0,C 180,E1 26246.551,E2 26246.551} C_VEL
LIN {X 0,Y 281.066,Z 1158.081,A -85,B 0,C 180,E1 26252.119,E2 26252.119} C_VEL
LIN {X 0,Y 281.266,Z 1157.555,A -85,B 0,C 180,E1 26252.575,E2 26252.575} C_VEL
LIN {X 0,Y 242.321,Z 1171.783,A -85,B 0,C 180,E1 26265.555,E2 26265.555} C_VEL
LIN {X 0,Y 220.79,Z 1179.04,A -85,B 0,C 180,E1 26279.999,E2 26279.999} C_VEL
LIN {X 0,Y 212.068,Z 1180.609,A -85,B 0,C 180,E1 26292.341,E2 26292.341} C_VEL
LIN {X 0,Y 209.199,Z 1179.737,A -85,B 0,C 180,E1 26301.168,E2 26301.168} C_VEL
LIN {X 0,Y 209.499,Z 1175.534,A -85,B 0,C 180,E1 26312.546,E2 26312.546} C_VEL
LIN {X 0,Y 212.985,Z 1168.884,A -85,B 0,C 180,E1 26322.67,E2 26322.67} C_VEL
LIN {X 0,Y 220.628,Z 1157.28,A -85,B 0,C 180,E1 26334.039,E2 26334.039} C_VEL
LIN {X 0,Y 231.693,Z 1143.527,A -85,B 0,C 180,E1 26343.16,E2 26343.16} C_VEL
LIN {X 0,Y 234.094,Z 1137.366,A -85,B 0,C 180,E1 26347.159,E2 26347.159} C_VEL
LIN {X 0,Y 237.228,Z 1130.509,A -85,B 0,C 180,E1 26351.017,E2 26351.017} C_VEL
LIN {X 0,Y 260.604,Z 1103.335,A -85,B 0,C 180,E1 26360.279,E2 26360.279} C_VEL
LIN {X 0,Y 284.825,Z 1072.473,A -85,B 0,C 180,E1 26367.196,E2 26367.196} C_VEL
LIN {X 0,Y 309.663,Z 1037.224,A -85,B 0,C 180,E1 26372.59,E2 26372.59} C_VEL
LIN {X 0,Y 310.934,Z 1034.252,A -85,B 0,C 180,E1 26373.145,E2 26373.145} C_VEL
LIN {X 0,Y 311.242,Z 1016.026,A -85,B 0,C 180,E1 26379.09,E2 26379.09} C_VEL
LIN {X 0,Y 309.875,Z 1000.23,A -85,B 0,C 180,E1 26385.047,E2 26385.047} C_VEL
LIN {X 0,Y 307.314,Z 985.849,A -85,B 0,C 180,E1 26391.57,E2 26391.57} C_VEL
LIN {X 0,Y 304.254,Z 973.878,A -85,B 0,C 180,E1 26398.577,E2 26398.577} C_VEL
LIN {X 0,Y 301.479,Z 963.64,A -85,B 0,C 180,E1 26406.689,E2 26406.689} C_VEL
LIN {X 0,Y 299.76,Z 957.363,A -85,B 0,C 180,E1 26415.116,E2 26415.116} C_VEL
LIN {X 0,Y 299.657,Z 955.43,A -85,B 0,C 180,E1 26423.806,E2 26423.806} C_VEL
LIN {X 0,Y 302.46,Z 956.862,A -85,B 0,C 180,E1 26433.283,E2 26433.283} C_VEL
LIN {X 0,Y 305.73,Z 961.467,A -85,B 0,C 180,E1 26439.928,E2 26439.928} C_VEL
LIN {X 0,Y 309.073,Z 966.533,A -85,B 0,C 180,E1 26444.947,E2 26444.947} C_VEL
LIN {X 0,Y 315.107,Z 977.466,A -85,B 0,C 180,E1 26452.377,E2 26452.377} C_VEL
LIN {X 0,Y 321.649,Z 992.778,A -85,B 0,C 180,E1 26459.423,E2 26459.423} C_VEL
LIN {X 0,Y 328.838,Z 1012.589,A -85,B 0,C 180,E1 26466.597,E2 26466.597} C_VEL
LIN {X 0,Y 335.899,Z 1036.687,A -85,B 0,C 180,E1 26473.613,E2 26473.613} C_VEL
LIN {X 0,Y 336.757,Z 1040.494,A -85,B 0,C 180,E1 26474.606,E2 26474.606} C_VEL
LIN {X 0,Y 315.225,Z 1079.396,A -85,B 0,C 180,E1 26477.986,E2 26477.986} C_VEL
LIN {X 0,Y 290.045,Z 1118.183,A -85,B 0,C 180,E1 26482.69,E2 26482.69} C_VEL
LIN {X 0,Y 262.399,Z 1155.692,A -85,B 0,C 180,E1 26489.555,E2 26489.555} C_VEL
LIN {X 0,Y 239.123,Z 1184.958,A -85,B 0,C 180,E1 26497.801,E2 26497.801} C_VEL
LIN {X 0,Y 220.616,Z 1208.385,A -85,B 0,C 180,E1 26507.722,E2 26507.722} C_VEL
LIN {X 0,Y 208.129,Z 1226.199,A -85,B 0,C 180,E1 26519.436,E2 26519.436} C_VEL
LIN {X 0,Y 202.931,Z 1236.964,A -85,B 0,C 180,E1 26530.404,E2 26530.404} C_VEL
LIN {X 0,Y 201.91,Z 1241.191,A -85,B 0,C 180,E1 26537.008,E2 26537.008} C_VEL
LIN {X 0,Y 202.073,Z 1244.123,A -85,B 0,C 180,E1 26545.694,E2 26545.694} C_VEL
LIN {X 0,Y 202.757,Z 1244.53,A -85,B 0,C 180,E1 26549.983,E2 26549.983} C_VEL
LIN {X 0,Y 201.917,Z 1242.462,A -85,B 0,C 180,E1 26558.59,E2 26558.59} C_VEL
LIN {X 0,Y 202.914,Z 1235.917,A -85,B 0,C 180,E1 26569.56,E2 26569.56} C_VEL
LIN {X 0,Y 209.599,Z 1222.719,A -85,B 0,C 180,E1 26582.711,E2 26582.711} C_VEL
LIN {X 0,Y 227.806,Z 1201.061,A -85,B 0,C 180,E1 26596.833,E2 26596.833} C_VEL
LIN {X 0,Y 269.976,Z 1164.308,A -85,B 0,C 180,E1 26611.915,E2 26611.915} C_VEL
LIN {X 0,Y 271.52,Z 1162.807,A -85,B 0,C 180,E1 26612.691,E2 26612.691} C_VEL
LIN {X 0,Y 234.001,Z 1174.927,A -85,B 0,C 180,E1 26625.546,E2 26625.546} C_VEL
LIN {X 0,Y 212.874,Z 1181.038,A -85,B 0,C 180,E1 26639.998,E2 26639.998} C_VEL
LIN {X 0,Y 204.004,Z 1182.12,A -85,B 0,C 180,E1 26652.837,E2 26652.837} C_VEL
LIN {X 0,Y 200.951,Z 1179.32,A -85,B 0,C 180,E1 26666.816,E2 26666.816} C_VEL
LIN {X 0,Y 203.325,Z 1173.533,A -85,B 0,C 180,E1 26678.147,E2 26678.147} C_VEL
LIN {X 0,Y 208.985,Z 1164.314,A -85,B 0,C 180,E1 26689.425,E2 26689.425} C_VEL
LIN {X 0,Y 220.966,Z 1149.167,A -85,B 0,C 180,E1 26701.419,E2 26701.419} C_VEL
LIN {X 0,Y 237.228,Z 1130.509,A -85,B 0,C 180,E1 26711.017,E2 26711.017} C_VEL
LIN {X 0,Y 241.013,Z 1123.165,A -85,B 0,C 180,E1 26714.708,E2 26714.708} C_VEL
LIN {X 0,Y 245.499,Z 1115.128,A -85,B 0,C 180,E1 26718.245,E2 26718.245} C_VEL
LIN {X 0,Y 270.469,Z 1085.365,A -85,B 0,C 180,E1 26726.025,E2 26726.025} C_VEL
LIN {X 0,Y 295.616,Z 1052.073,A -85,B 0,C 180,E1 26731.88,E2 26731.88} C_VEL
LIN {X 0,Y 304.723,Z 1038.788,A -85,B 0,C 180,E1 26733.698,E2 26733.698} C_VEL
LIN {X 0,Y 305.661,Z 1022.025,A -85,B 0,C 180,E1 26739.185,E2 26739.185} C_VEL
LIN {X 0,Y 304.684,Z 1006.527,A -85,B 0,C 180,E1 26745.104,E2 26745.104} C_VEL
LIN {X 0,Y 302.461,Z 991.782,A -85,B 0,C 180,E1 26751.923,E2 26751.923} C_VEL
LIN {X 0,Y 299.641,Z 979.673,A -85,B 0,C 180,E1 26759.238,E2 26759.238} C_VEL
LIN {X 0,Y 297.723,Z 971.549,A -85,B 0,C 180,E1 26765.708,E2 26765.708} C_VEL
LIN {X 0,Y 296.433,Z 966.526,A -85,B 0,C 180,E1 26771.519,E2 26771.519} C_VEL
LIN {X 0,Y 295.76,Z 963.226,A -85,B 0,C 180,E1 26778.385,E2 26778.385} C_VEL
LIN {X 0,Y 296.301,Z 962.46,A -85,B 0,C 180,E1 26785.88,E2 26785.88} C_VEL
LIN {X 0,Y 299.696,Z 964.869,A -85,B 0,C 180,E1 26795.196,E2 26795.196} C_VEL
LIN {X 0,Y 304.431,Z 971.763,A -85,B 0,C 180,E1 26803.521,E2 26803.521} C_VEL
LIN {X 0,Y 310.599,Z 983.152,A -85,B 0,C 180,E1 26811.609,E2 26811.609} C_VEL
LIN {X 0,Y 316.304,Z 997.059,A -85,B 0,C 180,E1 26818.338,E2 26818.338} C_VEL
LIN {X 0,Y 322.96,Z 1015.734,A -85,B 0,C 180,E1 26825.37,E2 26825.37} C_VEL
LIN {X 0,Y 329.421,Z 1038.274,A -85,B 0,C 180,E1 26832.249,E2 26832.249} C_VEL
LIN {X 0,Y 330.739,Z 1043.901,A -85,B 0,C 180,E1 26833.813,E2 26833.813} C_VEL
LIN {X 0,Y 305.683,Z 1086.836,A -85,B 0,C 180,E1 26837.619,E2 26837.619} C_VEL
LIN {X 0,Y 276.925,Z 1128.67,A -85,B 0,C 180,E1 26843.213,E2 26843.213} C_VEL
LIN {X 0,Y 251.031,Z 1161.959,A -85,B 0,C 180,E1 26850.057,E2 26850.057} C_VEL
LIN {X 0,Y 227.935,Z 1189.927,A -85,B 0,C 180,E1 26858.791,E2 26858.791} C_VEL
LIN {X 0,Y 209.752,Z 1212.141,A -85,B 0,C 180,E1 26869.56,E2 26869.56} C_VEL
LIN {X 0,Y 198.858,Z 1228.051,A -85,B 0,C 180,E1 26881.391,E2 26881.391} C_VEL
LIN {X 0,Y 194.723,Z 1237.028,A -85,B 0,C 180,E1 26891.898,E2 26891.898} C_VEL
LIN {X 0,Y 193.947,Z 1241.523,A -85,B 0,C 180,E1 26901.017,E2 26901.017} C_VEL
LIN {X 0,Y 194.961,Z 1243.176,A -85,B 0,C 180,E1 26909.982,E2 26909.982} C_VEL
LIN {X 0,Y 194.117,Z 1241.092,A -85,B 0,C 180,E1 26918.938,E2 26918.938} C_VEL
LIN {X 0,Y 195.169,Z 1234.818,A -85,B 0,C 180,E1 26930.107,E2 26930.107} C_VEL
LIN {X 0,Y 202.215,Z 1222.047,A -85,B 0,C 180,E1 26943.588,E2 26943.588} C_VEL
LIN {X 0,Y 222.115,Z 1200.285,A -85,B 0,C 180,E1 26958.422,E2 26958.422} C_VEL
LIN {X 0,Y 262.36,Z 1167.651,A -85,B 0,C 180,E1 26972.564,E2 26972.564} C_VEL
LIN {X 0,Y 220.682,Z 1179.392,A -85,B 0,C 180,E1 26988.145,E2 26988.145} C_VEL
LIN {X 0,Y 204.953,Z 1183.036,A -85,B 0,C 180,E1 26999.998,E2 26999.998} C_VEL
LIN {X 0,Y 195.95,Z 1183.623,A -85,B 0,C 180,E1 27013.374,E2 27013.374} C_VEL
LIN {X 0,Y 193.293,Z 1181.752,A -85,B 0,C 180,E1 27023.006,E2 27023.006} C_VEL
LIN {X 0,Y 193.932,Z 1177.801,A -85,B 0,C 180,E1 27033.05,E2 27033.05} C_VEL
LIN {X 0,Y 198.105,Z 1170.358,A -85,B 0,C 180,E1 27044.458,E2 27044.458} C_VEL
LIN {X 0,Y 207.407,Z 1157.789,A -85,B 0,C 180,E1 27056.91,E2 27056.91} C_VEL
LIN {X 0,Y 222.62,Z 1140.572,A -85,B 0,C 180,E1 27067.859,E2 27067.859} C_VEL
LIN {X 0,Y 244.841,Z 1115.861,A -85,B 0,C 180,E1 27078.004,E2 27078.004} C_VEL
LIN {X 0,Y 245.499,Z 1115.128,A -85,B 0,C 180,E1 27078.245,E2 27078.245} C_VEL
LIN {X 0,Y 250.392,Z 1106.59,A -85,B 0,C 180,E1 27081.611,E2 27081.611} C_VEL
LIN {X 0,Y 254.88,Z 1098.719,A -85,B 0,C 180,E1 27084.43,E2 27084.43} C_VEL
LIN {X 0,Y 255.957,Z 1097.446,A -85,B 0,C 180,E1 27084.752,E2 27084.752} C_VEL
LIN {X 0,Y 281.505,Z 1065.696,A -85,B 0,C 180,E1 27091.158,E2 27091.158} C_VEL
LIN {X 0,Y 298.526,Z 1042.106,A -85,B 0,C 180,E1 27094.6,E2 27094.6} C_VEL
LIN {X 0,Y 299.941,Z 1028.608,A -85,B 0,C 180,E1 27099.07,E2 27099.07} C_VEL
LIN {X 0,Y 299.632,Z 1014.16,A -85,B 0,C 180,E1 27104.617,E2 27104.617} C_VEL
LIN {X 0,Y 297.878,Z 999.346,A -85,B 0,C 180,E1 27111.44,E2 27111.44} C_VEL
LIN {X 0,Y 295.502,Z 987.294,A -85,B 0,C 180,E1 27118.642,E2 27118.642} C_VEL
LIN {X 0,Y 293.545,Z 977.836,A -85,B 0,C 180,E1 27126.296,E2 27126.296} C_VEL
LIN {X 0,Y 292.192,Z 972.122,A -85,B 0,C 180,E1 27133.618,E2 27133.618} C_VEL
LIN {X 0,Y 292.052,Z 969.586,A -85,B 0,C 180,E1 27141.624,E2 27141.624} C_VEL
LIN {X 0,Y 294.08,Z 970.266,A -85,B 0,C 180,E1 27150.892,E2 27150.892} C_VEL
LIN {X 0,Y 297.229,Z 973.68,A -85,B 0,C 180,E1 27157.927,E2 27157.927} C_VEL
LIN {X 0,Y 300.827,Z 979.237,A -85,B 0,C 180,E1 27163.877,E2 27163.877} C_VEL
LIN {X 0,Y 306.49,Z 989.94,A -85,B 0,C 180,E1 27171.496,E2 27171.496} C_VEL
LIN {X 0,Y 312.225,Z 1004.619,A -85,B 0,C 180,E1 27178.615,E2 27178.615} C_VEL
LIN {X 0,Y 318.257,Z 1022.669,A -85,B 0,C 180,E1 27185.45,E2 27185.45} C_VEL
LIN {X 0,Y 324.322,Z 1045.408,A -85,B 0,C 180,E1 27192.444,E2 27192.444} C_VEL
LIN {X 0,Y 324.581,Z 1047.357,A -85,B 0,C 180,E1 27192.947,E2 27192.947} C_VEL
LIN {X 0,Y 299.683,Z 1088.35,A -85,B 0,C 180,E1 27196.622,E2 27196.622} C_VEL
LIN {X 0,Y 271.163,Z 1128.781,A -85,B 0,C 180,E1 27202.085,E2 27202.085} C_VEL
LIN {X 0,Y 243.061,Z 1163.76,A -85,B 0,C 180,E1 27209.472,E2 27209.472} C_VEL
LIN {X 0,Y 220.5,Z 1190.104,A -85,B 0,C 180,E1 27218.08,E2 27218.08} C_VEL
LIN {X 0,Y 201.994,Z 1211.877,A -85,B 0,C 180,E1 27229.091,E2 27229.091} C_VEL
LIN {X 0,Y 190.781,Z 1227.669,A -85,B 0,C 180,E1 27241.605,E2 27241.605} C_VEL
LIN {X 0,Y 186.644,Z 1236.869,A -85,B 0,C 180,E1 27253.52,E2 27253.52} C_VEL
LIN {X 0,Y 186.458,Z 1241.295,A -85,B 0,C 180,E1 27265.333,E2 27265.333} C_VEL
LIN {X 0,Y 187.176,Z 1241.798,A -85,B 0,C 180,E1 27269.981,E2 27269.981} C_VEL
LIN {X 0,Y 186.281,Z 1239.747,A -85,B 0,C 180,E1 27279.317,E2 27279.317} C_VEL
LIN {X 0,Y 187.465,Z 1233.655,A -85,B 0,C 180,E1 27290.799,E2 27290.799} C_VEL
LIN {X 0,Y 195.169,Z 1221.077,A -85,B 0,C 180,E1 27304.827,E2 27304.827} C_VEL
LIN {X 0,Y 218.458,Z 1198.024,A -85,B 0,C 180,E1 27321.003,E2 27321.003} C_VEL
LIN {X 0,Y 252.163,Z 1172.343,A -85,B 0,C 180,E1 27332.842,E2 27332.842} C_VEL
LIN {X 0,Y 213.133,Z 1181.981,A -85,B 0,C 180,E1 27347.719,E2 27347.719} C_VEL
LIN {X 0,Y 196.386,Z 1185.168,A -85,B 0,C 180,E1 27360.639,E2 27360.639} C_VEL
LIN {X 0,Y 187.49,Z 1184.824,A -85,B 0,C 180,E1 27374.808,E2 27374.808} C_VEL
LIN {X 0,Y 185.484,Z 1180.8,A -85,B 0,C 180,E1 27389.258,E2 27389.258} C_VEL
LIN {X 0,Y 188.85,Z 1174.113,A -85,B 0,C 180,E1 27401.408,E2 27401.408} C_VEL
LIN {X 0,Y 196.394,Z 1163.503,A -85,B 0,C 180,E1 27413.785,E2 27413.785} C_VEL
LIN {X 0,Y 211.702,Z 1146.117,A -85,B 0,C 180,E1 27426.448,E2 27426.448} C_VEL
LIN {X 0,Y 231.646,Z 1124.822,A -85,B 0,C 180,E1 27436.445,E2 27436.445} C_VEL
LIN {X 0,Y 255.957,Z 1097.446,A -85,B 0,C 180,E1 27444.752,E2 27444.752} C_VEL
LIN {X 0,Y 260.849,Z 1090.153,A -85,B 0,C 180,E1 27446.913,E2 27446.913} C_VEL
LIN {X 0,Y 266.929,Z 1079.017,A -85,B 0,C 180,E1 27450.232,E2 27450.232} C_VEL
LIN {X 0,Y 267.983,Z 1077.598,A -85,B 0,C 180,E1 27450.516,E2 27450.516} C_VEL
LIN {X 0,Y 292.771,Z 1044.827,A -85,B 0,C 180,E1 27455.613,E2 27455.613} C_VEL
LIN {X 0,Y 294.258,Z 1031.424,A -85,B 0,C 180,E1 27460.25,E2 27460.25} C_VEL
LIN {X 0,Y 294.08,Z 1016.923,A -85,B 0,C 180,E1 27466.155,E2 27466.155} C_VEL
LIN {X 0,Y 292.761,Z 1003.686,A -85,B 0,C 180,E1 27472.646,E2 27472.646} C_VEL
LIN {X 0,Y 290.672,Z 992.044,A -85,B 0,C 180,E1 27480.034,E2 27480.034} C_VEL
LIN {X 0,Y 289.175,Z 984.124,A -85,B 0,C 180,E1 27486.73,E2 27486.73} C_VEL
LIN {X 0,Y 288.285,Z 979.359,A -85,B 0,C 180,E1 27492.969,E2 27492.969} C_VEL
LIN {X 0,Y 288.041,Z 976.512,A -85,B 0,C 180,E1 27500.989,E2 27500.989} C_VEL
LIN {X 0,Y 289.423,Z 976.702,A -85,B 0,C 180,E1 27508.53,E2 27508.53} C_VEL
LIN {X 0,Y 292.385,Z 979.034,A -85,B 0,C 180,E1 27515.581,E2 27515.581} C_VEL
LIN {X 0,Y 296.756,Z 985.901,A -85,B 0,C 180,E1 27523.65,E2 27523.65} C_VEL
LIN {X 0,Y 302.204,Z 996.581,A -85,B 0,C 180,E1 27531.374,E2 27531.374} C_VEL
LIN {X 0,Y 307.799,Z 1011.411,A -85,B 0,C 180,E1 27538.595,E2 27538.595} C_VEL
LIN {X 0,Y 313.814,Z 1030.661,A -85,B 0,C 180,E1 27545.874,E2 27545.874} C_VEL
LIN {X 0,Y 318.507,Z 1049.761,A -85,B 0,C 180,E1 27551.854,E2 27551.854} C_VEL
LIN {X 0,Y 295.027,Z 1087.995,A -85,B 0,C 180,E1 27555.389,E2 27555.389} C_VEL
LIN {X 0,Y 266.565,Z 1127.51,A -85,B 0,C 180,E1 27560.683,E2 27560.683} C_VEL
LIN {X 0,Y 237.711,Z 1162.467,A -85,B 0,C 180,E1 27568.049,E2 27568.049} C_VEL
LIN {X 0,Y 214.312,Z 1188.841,A -85,B 0,C 180,E1 27576.738,E2 27576.738} C_VEL
LIN {X 0,Y 194.175,Z 1211.667,A -85,B 0,C 180,E1 27588.655,E2 27588.655} C_VEL
LIN {X 0,Y 182.847,Z 1227.008,A -85,B 0,C 180,E1 27601.607,E2 27601.607} C_VEL
LIN {X 0,Y 178.923,Z 1235.302,A -85,B 0,C 180,E1 27612.787,E2 27612.787} C_VEL
LIN {X 0,Y 178.325,Z 1238.546,A -85,B 0,C 180,E1 27620.223,E2 27620.223} C_VEL
LIN {X 0,Y 179.38,Z 1240.351,A -85,B 0,C 180,E1 27629.98,E2 27629.98} C_VEL
LIN {X 0,Y 178.436,Z 1238.375,A -85,B 0,C 180,E1 27639.731,E2 27639.731} C_VEL
LIN {X 0,Y 179.315,Z 1233.668,A -85,B 0,C 180,E1 27649.678,E2 27649.678} C_VEL
LIN {X 0,Y 186.725,Z 1221.871,A -85,B 0,C 180,E1 27664.481,E2 27664.481} C_VEL
LIN {X 0,Y 209.314,Z 1200.614,A -85,B 0,C 180,E1 27680.918,E2 27680.918} C_VEL
LIN {X 0,Y 239.527,Z 1178.817,A -85,B 0,C 180,E1 27691.997,E2 27691.997} C_VEL
LIN {X 0,Y 241.606,Z 1176.972,A -85,B 0,C 180,E1 27693.151,E2 27693.151} C_VEL
LIN {X 0,Y 205.612,Z 1184.576,A -85,B 0,C 180,E1 27707.262,E2 27707.262} C_VEL
LIN {X 0,Y 189.004,Z 1186.975,A -85,B 0,C 180,E1 27719.998,E2 27719.998} C_VEL
LIN {X 0,Y 179.762,Z 1186.203,A -85,B 0,C 180,E1 27734.604,E2 27734.604} C_VEL
LIN {X 0,Y 177.838,Z 1181.534,A -85,B 0,C 180,E1 27750.647,E2 27750.647} C_VEL
LIN {X 0,Y 181.17,Z 1175.221,A -85,B 0,C 180,E1 27761.85,E2 27761.85} C_VEL
LIN {X 0,Y 189.292,Z 1164.207,A -85,B 0,C 180,E1 27774.884,E2 27774.884} C_VEL
LIN {X 0,Y 205.292,Z 1146.808,A -85,B 0,C 180,E1 27787.747,E2 27787.747} C_VEL
LIN {X 0,Y 226.263,Z 1125.036,A -85,B 0,C 180,E1 27797.972,E2 27797.972} C_VEL
LIN {X 0,Y 252.568,Z 1096.173,A -85,B 0,C 180,E1 27806.584,E2 27806.584} C_VEL
LIN {X 0,Y 267.983,Z 1077.598,A -85,B 0,C 180,E1 27810.516,E2 27810.516} C_VEL
LIN {X 0,Y 274.52,Z 1066.966,A -85,B 0,C 180,E1 27813.127,E2 27813.127} C_VEL
LIN {X 0,Y 281.201,Z 1055.774,A -85,B 0,C 180,E1 27815.543,E2 27815.543} C_VEL
LIN {X 0,Y 287.456,Z 1046.903,A -85,B 0,C 180,E1 27816.805,E2 27816.805} C_VEL
LIN {X 0,Y 288.859,Z 1030.373,A -85,B 0,C 180,E1 27823.072,E2 27823.072} C_VEL
LIN {X 0,Y 288.282,Z 1015.204,A -85,B 0,C 180,E1 27829.931,E2 27829.931} C_VEL
LIN {X 0,Y 286.96,Z 1003.785,A -85,B 0,C 180,E1 27836.477,E2 27836.477} C_VEL
LIN {X 0,Y 285.386,Z 993.668,A -85,B 0,C 180,E1 27844.065,E2 27844.065} C_VEL
LIN {X 0,Y 284.201,Z 986.781,A -85,B 0,C 180,E1 27851.9,E2 27851.9} C_VEL
LIN {X 0,Y 284.029,Z 983.51,A -85,B 0,C 180,E1 27860.33,E2 27860.33} C_VEL
LIN {X 0,Y 285.329,Z 983.457,A -85,B 0,C 180,E1 27868.026,E2 27868.026} C_VEL
LIN {X 0,Y 288.173,Z 985.685,A -85,B 0,C 180,E1 27875.2,E2 27875.2} C_VEL
LIN {X 0,Y 292.576,Z 992.568,A -85,B 0,C 180,E1 27883.499,E2 27883.499} C_VEL
LIN {X 0,Y 297.911,Z 1003.233,A -85,B 0,C 180,E1 27891.249,E2 27891.249} C_VEL
LIN {X 0,Y 303.141,Z 1018.081,A -85,B 0,C 180,E1 27898.572,E2 27898.572} C_VEL
LIN {X 0,Y 308.549,Z 1036.465,A -85,B 0,C 180,E1 27905.622,E2 27905.622} C_VEL
LIN {X 0,Y 312.41,Z 1053.151,A -85,B 0,C 180,E1 27910.98,E2 27910.98} C_VEL
LIN {X 0,Y 283.852,Z 1097.134,A -85,B 0,C 180,E1 27915.187,E2 27915.187} C_VEL
LIN {X 0,Y 255.729,Z 1133.881,A -85,B 0,C 180,E1 27920.591,E2 27920.591} C_VEL
LIN {X 0,Y 228.431,Z 1165.752,A -85,B 0,C 180,E1 27927.815,E2 27927.815} C_VEL
LIN {X 0,Y 202.124,Z 1194.214,A -85,B 0,C 180,E1 27938.255,E2 27938.255} C_VEL
LIN {X 0,Y 183.976,Z 1214.146,A -85,B 0,C 180,E1 27950.254,E2 27950.254} C_VEL
LIN {X 0,Y 173.619,Z 1228.43,A -85,B 0,C 180,E1 27964.182,E2 27964.182} C_VEL
LIN {X 0,Y 170.633,Z 1235.996,A -85,B 0,C 180,E1 27976.933,E2 27976.933} C_VEL
LIN {X 0,Y 170.821,Z 1238.439,A -85,B 0,C 180,E1 27984.904,E2 27984.904} C_VEL
LIN {X 0,Y 171.591,Z 1238.91,A -85,B 0,C 180,E1 27989.979,E2 27989.979} C_VEL
LIN {X 0,Y 170.58,Z 1237.033,A -85,B 0,C 180,E1 28000.184,E2 28000.184} C_VEL
LIN {X 0,Y 171.656,Z 1232.333,A -85,B 0,C 180,E1 28010.594,E2 28010.594} C_VEL
LIN {X 0,Y 179.873,Z 1220.694,A -85,B 0,C 180,E1 28025.994,E2 28025.994} C_VEL
LIN {X 0,Y 204.022,Z 1200.161,A -85,B 0,C 180,E1 28042.738,E2 28042.738} C_VEL
LIN {X 0,Y 232.541,Z 1180.861,A -85,B 0,C 180,E1 28052.944,E2 28052.944} C_VEL
LIN {X 0,Y 191.511,Z 1187.92,A -85,B 0,C 180,E1 28070.919,E2 28070.919} C_VEL
LIN {X 0,Y 177.061,Z 1188.73,A -85,B 0,C 180,E1 28084.894,E2 28084.894} C_VEL
LIN {X 0,Y 171.655,Z 1187.435,A -85,B 0,C 180,E1 28095.31,E2 28095.31} C_VEL
LIN {X 0,Y 170.269,Z 1181.978,A -85,B 0,C 180,E1 28112.169,E2 28112.169} C_VEL
LIN {X 0,Y 174.193,Z 1175.249,A -85,B 0,C 180,E1 28123.94,E2 28123.94} C_VEL
LIN {X 0,Y 183.603,Z 1163.333,A -85,B 0,C 180,E1 28137.494,E2 28137.494} C_VEL
LIN {X 0,Y 201.039,Z 1145.552,A -85,B 0,C 180,E1 28150.279,E2 28150.279} C_VEL
LIN {X 0,Y 225.093,Z 1121.085,A -85,B 0,C 180,E1 28161.038,E2 28161.038} C_VEL
LIN {X 0,Y 250.977,Z 1093.015,A -85,B 0,C 180,E1 28168.87,E2 28168.87} C_VEL
LIN {X 0,Y 280.239,Z 1057.073,A -85,B 0,C 180,E1 28175.356,E2 28175.356} C_VEL
LIN {X 0,Y 281.201,Z 1055.774,A -85,B 0,C 180,E1 28175.543,E2 28175.543} C_VEL
LIN {X 0,Y 283.157,Z 1050.714,A -85,B 0,C 180,E1 28176.877,E2 28176.877} C_VEL
LIN {X 0,Y 282.368,Z 1044.747,A -85,B 0,C 180,E1 28179.803,E2 28179.803} C_VEL
LIN {X 0,Y 283.312,Z 1030.919,A -85,B 0,C 180,E1 28185.479,E2 28185.479} C_VEL
LIN {X 0,Y 282.889,Z 1017.742,A -85,B 0,C 180,E1 28191.97,E2 28191.97} C_VEL
LIN {X 0,Y 281.669,Z 1006.805,A -85,B 0,C 180,E1 28198.884,E2 28198.884} C_VEL
LIN {X 0,Y 280.537,Z 997.942,A -85,B 0,C 180,E1 28206.349,E2 28206.349} C_VEL
LIN {X 0,Y 279.896,Z 993.04,A -85,B 0,C 180,E1 28212.696,E2 28212.696} C_VEL
LIN {X 0,Y 279.867,Z 990.4,A -85,B 0,C 180,E1 28219.62,E2 28219.62} C_VEL
LIN {X 0,Y 281.671,Z 990.515,A -85,B 0,C 180,E1 28229.154,E2 28229.154} C_VEL
LIN {X 0,Y 284.819,Z 993.534,A -85,B 0,C 180,E1 28236.757,E2 28236.757} C_VEL
LIN {X 0,Y 288.461,Z 999.352,A -85,B 0,C 180,E1 28243.447,E2 28243.447} C_VEL
LIN {X 0,Y 293.402,Z 1009.725,A -85,B 0,C 180,E1 28251.114,E2 28251.114} C_VEL
LIN {X 0,Y 298.485,Z 1024.763,A -85,B 0,C 180,E1 28258.549,E2 28258.549} C_VEL
LIN {X 0,Y 303.527,Z 1043.224,A -85,B 0,C 180,E1 28265.715,E2 28265.715} C_VEL
LIN {X 0,Y 306.301,Z 1055.995,A -85,B 0,C 180,E1 28269.943,E2 28269.943} C_VEL
LIN {X 0,Y 278.919,Z 1097.237,A -85,B 0,C 180,E1 28273.931,E2 28273.931} C_VEL
LIN {X 0,Y 248.823,Z 1135.414,A -85,B 0,C 180,E1 28279.604,E2 28279.604} C_VEL
LIN {X 0,Y 221.952,Z 1165.717,A -85,B 0,C 180,E1 28286.666,E2 28286.666} C_VEL
LIN {X 0,Y 195.918,Z 1192.933,A -85,B 0,C 180,E1 28296.822,E2 28296.822} C_VEL
LIN {X 0,Y 176.654,Z 1213.205,A -85,B 0,C 180,E1 28309.375,E2 28309.375} C_VEL
LIN {X 0,Y 166.282,Z 1226.657,A -85,B 0,C 180,E1 28322.952,E2 28322.952} C_VEL
LIN {X 0,Y 162.916,Z 1234.412,A -85,B 0,C 180,E1 28336.302,E2 28336.302} C_VEL
LIN {X 0,Y 162.999,Z 1236.921,A -85,B 0,C 180,E1 28344.659,E2 28344.659} C_VEL
LIN {X 0,Y 163.79,Z 1237.446,A -85,B 0,C 180,E1 28349.978,E2 28349.978} C_VEL
LIN {X 0,Y 162.769,Z 1235.686,A -85,B 0,C 180,E1 28360.678,E2 28360.678} C_VEL
LIN {X 0,Y 164.498,Z 1230.109,A -85,B 0,C 180,E1 28373.28,E2 28373.28} C_VEL
LIN {X 0,Y 176.134,Z 1216.955,A -85,B 0,C 180,E1 28390.511,E2 28390.511} C_VEL
LIN {X 0,Y 210.744,Z 1191.861,A -85,B 0,C 180,E1 28409.329,E2 28409.329} C_VEL
LIN {X 0,Y 222.147,Z 1184.87,A -85,B 0,C 180,E1 28413.234,E2 28413.234} C_VEL
LIN {X 0,Y 183.766,Z 1190.046,A -85,B 0,C 180,E1 28430.533,E2 28430.533} C_VEL
LIN {X 0,Y 167.51,Z 1190.035,A -85,B 0,C 180,E1 28447.297,E2 28447.297} C_VEL
LIN {X 0,Y 162.162,Z 1187.106,A -85,B 0,C 180,E1 28461.881,E2 28461.881} C_VEL
LIN {X 0,Y 163.475,Z 1181.121,A -85,B 0,C 180,E1 28476.582,E2 28476.582} C_VEL
LIN {X 0,Y 168.881,Z 1173.157,A -85,B 0,C 180,E1 28488.857,E2 28488.857} C_VEL
LIN {X 0,Y 181.697,Z 1158.945,A -85,B 0,C 180,E1 28503.138,E2 28503.138} C_VEL
LIN {X 0,Y 202.713,Z 1138.622,A -85,B 0,C 180,E1 28515.69,E2 28515.69} C_VEL
LIN {X 0,Y 228.457,Z 1112.788,A -85,B 0,C 180,E1 28525.38,E2 28525.38} C_VEL
LIN {X 0,Y 254.946,Z 1083.663,A -85,B 0,C 180,E1 28532.422,E2 28532.422} C_VEL
LIN {X 0,Y 281.397,Z 1050.335,A -85,B 0,C 180,E1 28537.728,E2 28537.728} C_VEL
LIN {X 0,Y 282.368,Z 1044.747,A -85,B 0,C 180,E1 28539.803,E2 28539.803} C_VEL
LIN {X 0,Y 281.169,Z 1040.393,A -85,B 0,C 180,E1 28542.311,E2 28542.311} C_VEL
LIN {X 0,Y 277.77,Z 1034.517,A -85,B 0,C 180,E1 28546.655,E2 28546.655} C_VEL
LIN {X 0,Y 277.606,Z 1021.624,A -85,B 0,C 180,E1 28553.374,E2 28553.374} C_VEL
LIN {X 0,Y 276.573,Z 1010.062,A -85,B 0,C 180,E1 28561.351,E2 28561.351} C_VEL
LIN {X 0,Y 275.855,Z 1002.711,A -85,B 0,C 180,E1 28568.332,E2 28568.332} C_VEL
LIN {X 0,Y 275.514,Z 998.393,A -85,B 0,C 180,E1 28575.496,E2 28575.496} C_VEL
LIN {X 0,Y 275.998,Z 996.786,A -85,B 0,C 180,E1 28582.973,E2 28582.973} C_VEL
LIN {X 0,Y 278.063,Z 997.57,A -85,B 0,C 180,E1 28590.723,E2 28590.723} C_VEL
LIN {X 0,Y 281.153,Z 1001.053,A -85,B 0,C 180,E1 28597.903,E2 28597.903} C_VEL
LIN {X 0,Y 284.048,Z 1005.831,A -85,B 0,C 180,E1 28603.288,E2 28603.288} C_VEL
LIN {X 0,Y 288.841,Z 1016.163,A -85,B 0,C 180,E1 28610.972,E2 28610.972} C_VEL
LIN {X 0,Y 293.154,Z 1029.627,A -85,B 0,C 180,E1 28617.786,E2 28617.786} C_VEL
LIN {X 0,Y 297.902,Z 1047.908,A -85,B 0,C 180,E1 28625.093,E2 28625.093} C_VEL
LIN {X 0,Y 299.968,Z 1059.708,A -85,B 0,C 180,E1 28629.057,E2 28629.057} C_VEL
LIN {X 0,Y 272.625,Z 1099.15,A -85,B 0,C 180,E1 28632.876,E2 28632.876} C_VEL
LIN {X 0,Y 242.317,Z 1136.561,A -85,B 0,C 180,E1 28638.494,E2 28638.494} C_VEL
LIN {X 0,Y 214.17,Z 1167.071,A -85,B 0,C 180,E1 28645.862,E2 28645.862} C_VEL
LIN {X 0,Y 189.535,Z 1191.933,A -85,B 0,C 180,E1 28655.448,E2 28655.448} C_VEL
LIN {X 0,Y 169.473,Z 1212.063,A -85,B 0,C 180,E1 28668.304,E2 28668.304} C_VEL
LIN {X 0,Y 158.173,Z 1226.167,A -85,B 0,C 180,E1 28683.405,E2 28683.405} C_VEL
LIN {X 0,Y 155.078,Z 1233.35,A -85,B 0,C 180,E1 28697.002,E2 28697.002} C_VEL
LIN {X 0,Y 155.995,Z 1236.003,A -85,B 0,C 180,E1 28709.977,E2 28709.977} C_VEL
LIN {X 0,Y 154.895,Z 1233.828,A -85,B 0,C 180,E1 28722.702,E2 28722.702} C_VEL
LIN {X 0,Y 157.695,Z 1227.73,A -85,B 0,C 180,E1 28736.455,E2 28736.455} C_VEL
LIN {X 0,Y 172.381,Z 1213.902,A -85,B 0,C 180,E1 28754.499,E2 28754.499} C_VEL
LIN {X 0,Y 209.638,Z 1189.903,A -85,B 0,C 180,E1 28772.321,E2 28772.321} C_VEL
LIN {X 0,Y 211.913,Z 1188.349,A -85,B 0,C 180,E1 28773.402,E2 28773.402} C_VEL
LIN {X 0,Y 175.973,Z 1192.095,A -85,B 0,C 180,E1 28790.11,E2 28790.11} C_VEL
LIN {X 0,Y 160.784,Z 1191.694,A -85,B 0,C 180,E1 28805.39,E2 28805.39} C_VEL
LIN {X 0,Y 155.374,Z 1189.614,A -85,B 0,C 180,E1 28816.96,E2 28816.96} C_VEL
LIN {X 0,Y 154.527,Z 1184.443,A -85,B 0,C 180,E1 28832.077,E2 28832.077} C_VEL
LIN {X 0,Y 159.159,Z 1176.951,A -85,B 0,C 180,E1 28845.679,E2 28845.679} C_VEL
LIN {X 0,Y 170.283,Z 1164.304,A -85,B 0,C 180,E1 28860.522,E2 28860.522} C_VEL
LIN {X 0,Y 189.161,Z 1146.48,A -85,B 0,C 180,E1 28873.438,E2 28873.438} C_VEL
LIN {X 0,Y 214.773,Z 1122.03,A -85,B 0,C 180,E1 28884.205,E2 28884.205} C_VEL
LIN {X 0,Y 241.885,Z 1093.865,A -85,B 0,C 180,E1 28891.898,E2 28891.898} C_VEL
LIN {X 0,Y 272.001,Z 1058.197,A -85,B 0,C 180,E1 28898.157,E2 28898.157} C_VEL
LIN {X 0,Y 275.931,Z 1052.44,A -85,B 0,C 180,E1 28899.084,E2 28899.084} C_VEL
LIN {X 0,Y 277.64,Z 1037.767,A -85,B 0,C 180,E1 28905.123,E2 28905.123} C_VEL
LIN {X 0,Y 277.77,Z 1034.517,A -85,B 0,C 180,E1 28906.655,E2 28906.655} C_VEL
LIN {X 0,Y 276.116,Z 1031.136,A -85,B 0,C 180,E1 28909.257,E2 28909.257} C_VEL
LIN {X 0,Y 272.361,Z 1027.205,A -85,B 0,C 180,E1 28913.757,E2 28913.757} C_VEL
LIN {X 0,Y 271.739,Z 1016.928,A -85,B 0,C 180,E1 28920.97,E2 28920.97} C_VEL
LIN {X 0,Y 271.304,Z 1008.952,A -85,B 0,C 180,E1 28928.768,E2 28928.768} C_VEL
LIN {X 0,Y 271.105,Z 1004.69,A -85,B 0,C 180,E1 28936.452,E2 28936.452} C_VEL
LIN {X 0,Y 271.659,Z 1003.548,A -85,B 0,C 180,E1 28942.28,E2 28942.28} C_VEL
LIN {X 0,Y 274.225,Z 1004.662,A -85,B 0,C 180,E1 28951.868,E2 28951.868} C_VEL
LIN {X 0,Y 276.946,Z 1007.864,A -85,B 0,C 180,E1 28958.088,E2 28958.088} C_VEL
LIN {X 0,Y 280.309,Z 1013.77,A -85,B 0,C 180,E1 28964.365,E2 28964.365} C_VEL
LIN {X 0,Y 284.636,Z 1023.703,A -85,B 0,C 180,E1 28971.516,E2 28971.516} C_VEL
LIN {X 0,Y 289.167,Z 1039.382,A -85,B 0,C 180,E1 28979.253,E2 28979.253} C_VEL
LIN {X 0,Y 293.31,Z 1058.198,A -85,B 0,C 180,E1 28986.525,E2 28986.525} C_VEL
LIN {X 0,Y 294.045,Z 1062.145,A -85,B 0,C 180,E1 28987.894,E2 28987.894} C_VEL
LIN {X 0,Y 264.953,Z 1102.891,A -85,B 0,C 180,E1 28992.017,E2 28992.017} C_VEL
LIN {X 0,Y 235.755,Z 1137.658,A -85,B 0,C 180,E1 28997.365,E2 28997.365} C_VEL
LIN {X 0,Y 205.058,Z 1169.755,A -85,B 0,C 180,E1 29005.446,E2 29005.446} C_VEL
LIN {X 0,Y 180.374,Z 1193.568,A -85,B 0,C 180,E1 29015.372,E2 29015.372} C_VEL
LIN {X 0,Y 160.574,Z 1212.853,A -85,B 0,C 180,E1 29028.836,E2 29028.836} C_VEL
LIN {X 0,Y 150.413,Z 1225.068,A -85,B 0,C 180,E1 29043.041,E2 29043.041} C_VEL
LIN {X 0,Y 147.223,Z 1232.406,A -85,B 0,C 180,E1 29058.13,E2 29058.13} C_VEL
LIN {X 0,Y 148.214,Z 1234.535,A -85,B 0,C 180,E1 29069.976,E2 29069.976} C_VEL
LIN {X 0,Y 147.107,Z 1232.946,A -85,B 0,C 180,E1 29081.83,E2 29081.83} C_VEL
LIN {X 0,Y 149.961,Z 1226.887,A -85,B 0,C 180,E1 29096.934,E2 29096.934} C_VEL
LIN {X 0,Y 166.456,Z 1212.896,A -85,B 0,C 180,E1 29116.539,E2 29116.539} C_VEL
LIN {X 0,Y 202.335,Z 1191.68,A -85,B 0,C 180,E1 29133.379,E2 29133.379} C_VEL
LIN {X 0,Y 168.188,Z 1194.145,A -85,B 0,C 180,E1 29149.647,E2 29149.647} C_VEL
LIN {X 0,Y 152.047,Z 1192.992,A -85,B 0,C 180,E1 29166.589,E2 29166.589} C_VEL
LIN {X 0,Y 146.264,Z 1188.583,A -85,B 0,C 180,E1 29184.405,E2 29184.405} C_VEL
LIN {X 0,Y 148.775,Z 1181.878,A -85,B 0,C 180,E1 29199.751,E2 29199.751} C_VEL
LIN {X 0,Y 156.804,Z 1171.812,A -85,B 0,C 180,E1 29214.704,E2 29214.704} C_VEL
LIN {X 0,Y 173.73,Z 1155.646,A -85,B 0,C 180,E1 29229.662,E2 29229.662} C_VEL
LIN {X 0,Y 198.422,Z 1133.21,A -85,B 0,C 180,E1 29241.859,E2 29241.859} C_VEL
LIN {X 0,Y 225.468,Z 1107.001,A -85,B 0,C 180,E1 29250.492,E2 29250.492} C_VEL
LIN {X 0,Y 254.917,Z 1074.776,A -85,B 0,C 180,E1 29257.2,E2 29257.2} C_VEL
LIN {X 0,Y 270.215,Z 1055.641,A -85,B 0,C 180,E1 29260.118,E2 29260.118} C_VEL
LIN {X 0,Y 272.03,Z 1041.637,A -85,B 0,C 180,E1 29266.139,E2 29266.139} C_VEL
LIN {X 0,Y 272.372,Z 1028.701,A -85,B 0,C 180,E1 29272.865,E2 29272.865} C_VEL
LIN {X 0,Y 272.361,Z 1027.205,A -85,B 0,C 180,E1 29273.757,E2 29273.757} C_VEL
LIN {X 0,Y 270.555,Z 1025.128,A -85,B 0,C 180,E1 29276.467,E2 29276.467} C_VEL
LIN {X 0,Y 266.84,Z 1023.173,A -85,B 0,C 180,E1 29281.108,E2 29281.108} C_VEL
LIN {X 0,Y 266.707,Z 1015.612,A -85,B 0,C 180,E1 29288.568,E2 29288.568} C_VEL
LIN {X 0,Y 266.583,Z 1012.826,A -85,B 0,C 180,E1 29292.876,E2 29292.876} C_VEL
LIN {X 0,Y 267.086,Z 1010.135,A -85,B 0,C 180,E1 29301.517,E2 29301.517} C_VEL
LIN {X 0,Y 269.069,Z 1010.653,A -85,B 0,C 180,E1 29309.643,E2 29309.643} C_VEL
LIN {X 0,Y 272.215,Z 1013.819,A -85,B 0,C 180,E1 29317.137,E2 29317.137} C_VEL
LIN {X 0,Y 275.674,Z 1020.012,A -85,B 0,C 180,E1 29324.096,E2 29324.096} C_VEL
LIN {X 0,Y 279.839,Z 1030.1,A -85,B 0,C 180,E1 29331.462,E2 29331.462} C_VEL
LIN {X 0,Y 284.072,Z 1045.763,A -85,B 0,C 180,E1 29339.239,E2 29339.239} C_VEL
LIN {X 0,Y 287.882,Z 1064.895,A -85,B 0,C 180,E1 29346.707,E2 29346.707} C_VEL
LIN {X 0,Y 275.081,Z 1083.577,A -85,B 0,C 180,E1 29348.514,E2 29348.514} C_VEL
LIN {X 0,Y 244.697,Z 1121.658,A -85,B 0,C 180,E1 29353.201,E2 29353.201} C_VEL
LIN {X 0,Y 213.105,Z 1155.483,A -85,B 0,C 180,E1 29359.983,E2 29359.983} C_VEL
LIN {X 0,Y 185.436,Z 1182.121,A -85,B 0,C 180,E1 29368.809,E2 29368.809} C_VEL
LIN {X 0,Y 161.146,Z 1204.215,A -85,B 0,C 180,E1 29381.364,E2 29381.364} C_VEL
LIN {X 0,Y 146.516,Z 1218.964,A -85,B 0,C 180,E1 29395.595,E2 29395.595} C_VEL
LIN {X 0,Y 140.116,Z 1228.414,A -85,B 0,C 180,E1 29411.097,E2 29411.097} C_VEL
LIN {X 0,Y 139.546,Z 1232.292,A -85,B 0,C 180,E1 29423.758,E2 29423.758} C_VEL
LIN {X 0,Y 140.411,Z 1233.085,A -85,B 0,C 180,E1 29429.975,E2 29429.975} C_VEL
LIN {X 0,Y 139.299,Z 1231.503,A -85,B 0,C 180,E1 29442.504,E2 29442.504} C_VEL
LIN {X 0,Y 142.617,Z 1225.599,A -85,B 0,C 180,E1 29458.447,E2 29458.447} C_VEL
LIN {X 0,Y 161.075,Z 1211.725,A -85,B 0,C 180,E1 29478.953,E2 29478.953} C_VEL
LIN {X 0,Y 190.037,Z 1195.753,A -85,B 0,C 180,E1 29492.744,E2 29492.744} C_VEL
LIN {X 0,Y 191.6,Z 1194.7,A -85,B 0,C 180,E1 29493.669,E2 29493.669} C_VEL
LIN {X 0,Y 154.033,Z 1195.814,A -85,B 0,C 180,E1 29514.368,E2 29514.368} C_VEL
LIN {X 0,Y 141.234,Z 1193.171,A -85,B 0,C 180,E1 29532.353,E2 29532.353} C_VEL
LIN {X 0,Y 138.526,Z 1188.004,A -85,B 0,C 180,E1 29549.286,E2 29549.286} C_VEL
LIN {X 0,Y 142.675,Z 1180.769,A -85,B 0,C 180,E1 29564.301,E2 29564.301} C_VEL
LIN {X 0,Y 153.723,Z 1168.56,A -85,B 0,C 180,E1 29580.588,E2 29580.588} C_VEL
LIN {X 0,Y 173.728,Z 1150.899,A -85,B 0,C 180,E1 29594.896,E2 29594.896} C_VEL
LIN {X 0,Y 198.914,Z 1128.455,A -85,B 0,C 180,E1 29605.661,E2 29605.661} C_VEL
LIN {X 0,Y 228.994,Z 1099.381,A -85,B 0,C 180,E1 29614.113,E2 29614.113} C_VEL
LIN {X 0,Y 260.211,Z 1064.18,A -85,B 0,C 180,E1 29620.407,E2 29620.407} C_VEL
LIN {X 0,Y 264.522,Z 1058.569,A -85,B 0,C 180,E1 29621.312,E2 29621.312} C_VEL
LIN {X 0,Y 266.478,Z 1045.471,A -85,B 0,C 180,E1 29627.202,E2 29627.202} C_VEL
LIN {X 0,Y 267.131,Z 1032.485,A -85,B 0,C 180,E1 29634.359,E2 29634.359} C_VEL
LIN {X 0,Y 266.84,Z 1023.173,A -85,B 0,C 180,E1 29641.108,E2 29641.108} C_VEL
LIN {X 0,Y 265.251,Z 1021.949,A -85,B 0,C 180,E1 29643.904,E2 29643.904} C_VEL
LIN {X 0,Y 261.858,Z 1021.943,A -85,B 0,C 180,E1 29648.68,E2 29648.68} C_VEL
LIN {X 0,Y 262.048,Z 1017.942,A -85,B 0,C 180,E1 29656.219,E2 29656.219} C_VEL
LIN {X 0,Y 263.182,Z 1016.607,A -85,B 0,C 180,E1 29664.963,E2 29664.963} C_VEL
LIN {X 0,Y 265.863,Z 1018.122,A -85,B 0,C 180,E1 29672.958,E2 29672.958} C_VEL
LIN {X 0,Y 269.273,Z 1022.637,A -85,B 0,C 180,E1 29680.326,E2 29680.326} C_VEL
LIN {X 0,Y 273.656,Z 1032.512,A -85,B 0,C 180,E1 29688.842,E2 29688.842} C_VEL
LIN {X 0,Y 277.073,Z 1044.674,A -85,B 0,C 180,E1 29695.751,E2 29695.751} C_VEL
LIN {X 0,Y 280.695,Z 1061.371,A -85,B 0,C 180,E1 29703.087,E2 29703.087} C_VEL
LIN {X 0,Y 281.773,Z 1068.276,A -85,B 0,C 180,E1 29705.772,E2 29705.772} C_VEL
LIN {X 0,Y 251.264,Z 1108.268,A -85,B 0,C 180,E1 29709.892,E2 29709.892} C_VEL
LIN {X 0,Y 217.433,Z 1145.405,A -85,B 0,C 180,E1 29716.141,E2 29716.141} C_VEL
LIN {X 0,Y 187.159,Z 1174.305,A -85,B 0,C 180,E1 29724.424,E2 29724.424} C_VEL
LIN {X 0,Y 159.824,Z 1198.474,A -85,B 0,C 180,E1 29736.485,E2 29736.485} C_VEL
LIN {X 0,Y 140.975,Z 1215.608,A -85,B 0,C 180,E1 29752.019,E2 29752.019} C_VEL
LIN {X 0,Y 133.207,Z 1225.307,A -85,B 0,C 180,E1 29767.131,E2 29767.131} C_VEL
LIN {X 0,Y 131.745,Z 1229.104,A -85,B 0,C 180,E1 29776.711,E2 29776.711} C_VEL
LIN {X 0,Y 132.622,Z 1231.616,A -85,B 0,C 180,E1 29789.973,E2 29789.973} C_VEL
LIN {X 0,Y 131.494,Z 1230.044,A -85,B 0,C 180,E1 29803.259,E2 29803.259} C_VEL
LIN {X 0,Y 135.383,Z 1224.318,A -85,B 0,C 180,E1 29820.119,E2 29820.119} C_VEL
LIN {X 0,Y 157.34,Z 1209.869,A -85,B 0,C 180,E1 29842.365,E2 29842.365} C_VEL
LIN {X 0,Y 179.62,Z 1198.562,A -85,B 0,C 180,E1 29852.777,E2 29852.777} C_VEL
LIN {X 0,Y 181,Z 1197.532,A -85,B 0,C 180,E1 29853.925,E2 29853.925} C_VEL
LIN {X 0,Y 146.029,Z 1197.445,A -85,B 0,C 180,E1 29874.059,E2 29874.059} C_VEL
LIN {X 0,Y 132.996,Z 1194.064,A -85,B 0,C 180,E1 29893.131,E2 29893.131} C_VEL
LIN {X 0,Y 130.853,Z 1188.338,A -85,B 0,C 180,E1 29911.188,E2 29911.188} C_VEL
LIN {X 0,Y 135.623,Z 1180.878,A -85,B 0,C 180,E1 29926.41,E2 29926.41} C_VEL
LIN {X 0,Y 147.858,Z 1168.452,A -85,B 0,C 180,E1 29943.03,E2 29943.03} C_VEL
LIN {X 0,Y 168.047,Z 1151.437,A -85,B 0,C 180,E1 29956.761,E2 29956.761} C_VEL
LIN {X 0,Y 196.51,Z 1126.714,A -85,B 0,C 180,E1 29968.288,E2 29968.288} C_VEL
LIN {X 0,Y 225.762,Z 1098.784,A -85,B 0,C 180,E1 29976.037,E2 29976.037} C_VEL
LIN {X 0,Y 257.302,Z 1063.803,A -85,B 0,C 180,E1 29982.073,E2 29982.073} C_VEL
LIN {X 0,Y 258.845,Z 1061.815,A -85,B 0,C 180,E1 29982.436,E2 29982.436} C_VEL
LIN {X 0,Y 261.039,Z 1048.832,A -85,B 0,C 180,E1 29988.579,E2 29988.579} C_VEL
LIN {X 0,Y 261.847,Z 1036.628,A -85,B 0,C 180,E1 29995.697,E2 29995.697} C_VEL
LIN {X 0,Y 261.987,Z 1026.324,A -85,B 0,C 180,E1 30003.863,E2 30003.863} C_VEL
LIN {X 0,Y 261.858,Z 1021.943,A -85,B 0,C 180,E1 30008.68,E2 30008.68} C_VEL
LIN {X 0,Y 260.371,Z 1022.071,A -85,B 0,C 180,E1 30011.535,E2 30011.535} C_VEL
LIN {X 0,Y 257.176,Z 1024.361,A -85,B 0,C 180,E1 30016.371,E2 30016.371} C_VEL
LIN {X 0,Y 258.679,Z 1023.098,A -85,B 0,C 180,E1 30024.888,E2 30024.888} C_VEL
LIN {X 0,Y 261.123,Z 1024.462,A -85,B 0,C 180,E1 30032.426,E2 30032.426} C_VEL
LIN {X 0,Y 264.478,Z 1028.816,A -85,B 0,C 180,E1 30039.955,E2 30039.955} C_VEL
LIN {X 0,Y 268.294,Z 1037.448,A -85,B 0,C 180,E1 30047.809,E2 30047.809} C_VEL
LIN {X 0,Y 271.414,Z 1048.539,A -85,B 0,C 180,E1 30054.512,E2 30054.512} C_VEL
LIN {X 0,Y 274.579,Z 1064.281,A -85,B 0,C 180,E1 30061.827,E2 30061.827} C_VEL
LIN {X 0,Y 275.643,Z 1071.146,A -85,B 0,C 180,E1 30064.588,E2 30064.588} C_VEL
LIN {X 0,Y 246.37,Z 1108.483,A -85,B 0,C 180,E1 30068.456,E2 30068.456} C_VEL
LIN {X 0,Y 212.114,Z 1145.186,A -85,B 0,C 180,E1 30074.587,E2 30074.587} C_VEL
LIN {X 0,Y 180.648,Z 1174.206,A -85,B 0,C 180,E1 30083.009,E2 30083.009} C_VEL
LIN {X 0,Y 154.941,Z 1196.044,A -85,B 0,C 180,E1 30093.968,E2 30093.968} C_VEL
LIN {X 0,Y 134.794,Z 1213.323,A -85,B 0,C 180,E1 30109.555,E2 30109.555} C_VEL
LIN {X 0,Y 125.7,Z 1223.642,A -85,B 0,C 180,E1 30126.014,E2 30126.014} C_VEL
LIN {X 0,Y 123.928,Z 1227.842,A -85,B 0,C 180,E1 30137.277,E2 30137.277} C_VEL
LIN {X 0,Y 124.807,Z 1230.153,A -85,B 0,C 180,E1 30149.972,E2 30149.972} C_VEL
LIN {X 0,Y 123.682,Z 1228.607,A -85,B 0,C 180,E1 30164.114,E2 30164.114} C_VEL
LIN {X 0,Y 128.277,Z 1223.069,A -85,B 0,C 180,E1 30181.978,E2 30181.978} C_VEL
LIN {X 0,Y 152.315,Z 1209.015,A -85,B 0,C 180,E1 30204.889,E2 30204.889} C_VEL
LIN {X 0,Y 171.312,Z 1199.999,A -85,B 0,C 180,E1 30213.83,E2 30213.83} C_VEL
LIN {X 0,Y 136.393,Z 1198.69,A -85,B 0,C 180,E1 30235.288,E2 30235.288} C_VEL
LIN {X 0,Y 124.654,Z 1194.9,A -85,B 0,C 180,E1 30254.245,E2 30254.245} C_VEL
LIN {X 0,Y 123.411,Z 1188.427,A -85,B 0,C 180,E1 30273.891,E2 30273.891} C_VEL
LIN {X 0,Y 128.599,Z 1181.177,A -85,B 0,C 180,E1 30288.426,E2 30288.426} C_VEL
LIN {X 0,Y 143.329,Z 1167.433,A -85,B 0,C 180,E1 30306.568,E2 30306.568} C_VEL
LIN {X 0,Y 168.084,Z 1147.223,A -85,B 0,C 180,E1 30321.42,E2 30321.42} C_VEL
LIN {X 0,Y 196.495,Z 1123.124,A -85,B 0,C 180,E1 30331.551,E2 30331.551} C_VEL
LIN {X 0,Y 229.768,Z 1090.956,A -85,B 0,C 180,E1 30339.461,E2 30339.461} C_VEL
LIN {X 0,Y 252.735,Z 1065.439,A -85,B 0,C 180,E1 30343.504,E2 30343.504} C_VEL
LIN {X 0,Y 255.231,Z 1054.466,A -85,B 0,C 180,E1 30348.704,E2 30348.704} C_VEL
LIN {X 0,Y 256.448,Z 1043.152,A -85,B 0,C 180,E1 30355.379,E2 30355.379} C_VEL
LIN {X 0,Y 256.832,Z 1033.416,A -85,B 0,C 180,E1 30363.097,E2 30363.097} C_VEL
LIN {X 0,Y 257.101,Z 1027.129,A -85,B 0,C 180,E1 30370.296,E2 30370.296} C_VEL
LIN {X 0,Y 257.176,Z 1024.361,A -85,B 0,C 180,E1 30376.371,E2 30376.371} C_VEL
LIN {X 0,Y 256.042,Z 1025.644,A -85,B 0,C 180,E1 30379.278,E2 30379.278} C_VEL
LIN {X 0,Y 253.685,Z 1029.517,A -85,B 0,C 180,E1 30384.152,E2 30384.152} C_VEL
LIN {X 0,Y 256.347,Z 1030.781,A -85,B 0,C 180,E1 30392.18,E2 30392.18} C_VEL
LIN {X 0,Y 260.107,Z 1035.934,A -85,B 0,C 180,E1 30400.792,E2 30400.792} C_VEL
LIN {X 0,Y 263.59,Z 1044.379,A -85,B 0,C 180,E1 30408.302,E2 30408.302} C_VEL
LIN {X 0,Y 266.517,Z 1056.015,A -85,B 0,C 180,E1 30415.123,E2 30415.123} C_VEL
LIN {X 0,Y 269.163,Z 1071.479,A -85,B 0,C 180,E1 30422.315,E2 30422.315} C_VEL
LIN {X 0,Y 269.561,Z 1074.207,A -85,B 0,C 180,E1 30423.415,E2 30423.415} C_VEL
LIN {X 0,Y 238.398,Z 1112.292,A -85,B 0,C 180,E1 30427.435,E2 30427.435} C_VEL
LIN {X 0,Y 205.672,Z 1146.161,A -85,B 0,C 180,E1 30433.233,E2 30433.233} C_VEL
LIN {X 0,Y 171.638,Z 1176.364,A -85,B 0,C 180,E1 30442.37,E2 30442.37} C_VEL
LIN {X 0,Y 145.675,Z 1197.301,A -85,B 0,C 180,E1 30453.876,E2 30453.876} C_VEL
LIN {X 0,Y 125.2,Z 1214.236,A -85,B 0,C 180,E1 30471.115,E2 30471.115} C_VEL
LIN {X 0,Y 117.503,Z 1223.054,A -85,B 0,C 180,E1 30487.275,E2 30487.275} C_VEL
LIN {X 0,Y 116.103,Z 1227.584,A -85,B 0,C 180,E1 30502.491,E2 30502.491} C_VEL
LIN {X 0,Y 117.006,Z 1228.664,A -85,B 0,C 180,E1 30509.97,E2 30509.97} C_VEL
